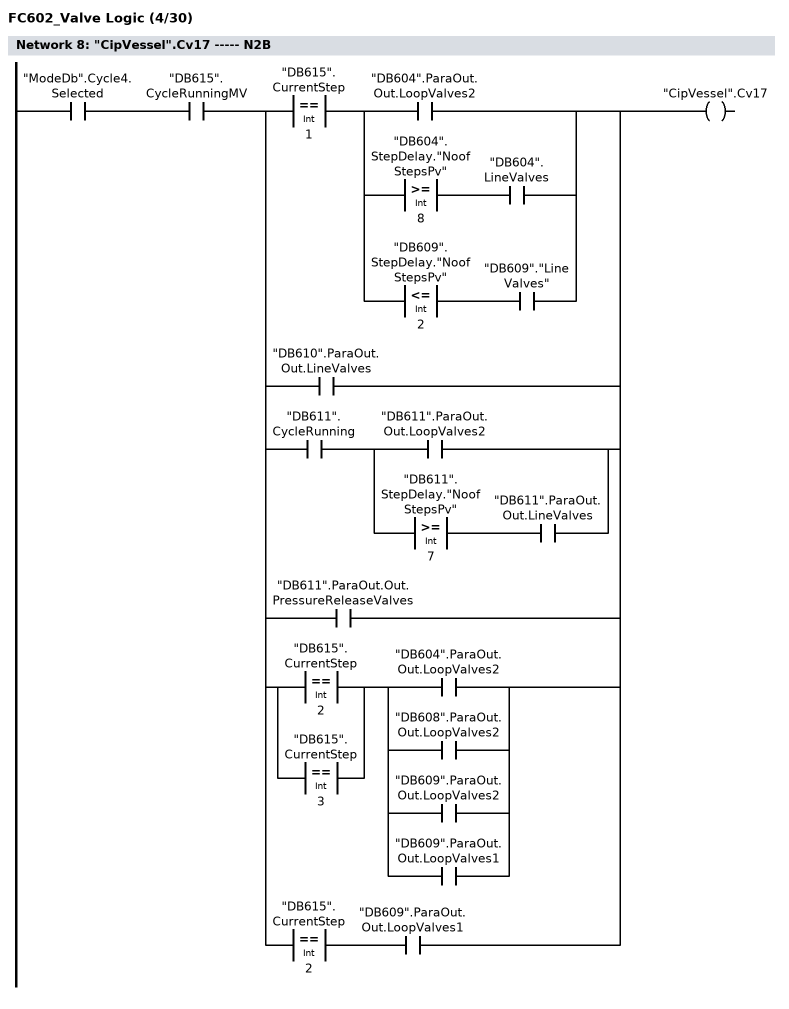
   RUNG wire#powerrail
      Contact( "ModeDb".Cycle4.Selected )
      Contact( "DB615".CycleRunningMV )
      wire#w1
      { S7_Templates := "SrcType := Int" } EQ_Contact(in1 := "DB615".CurrentStep, in2 := 1)
      wire#w2
      Contact( "DB604".ParaOut.Out.LoopValves2 )
      wire#w3
      Coil( "CipVessel".Cv17 )
   END_RUNG
   RUNG wire#w2
      { S7_Templates := "SrcType := Int" } GE_Contact(in1 := "DB604".StepDelay."Noof StepsPv", in2 := 8)
      Contact( "DB604".LineValves )
   END_RUNG wire#w3
   RUNG wire#w2
      { S7_Templates := "SrcType := Int" } LE_Contact(in1 := "DB609".StepDelay."Noof StepsPv", in2 := 2)
      Contact( "DB609"."Line Valves" )
   END_RUNG wire#w3
   RUNG wire#w1
      Contact( "DB610".ParaOut.Out.LineValves )
   END_RUNG wire#w3
   RUNG wire#w1
      Contact( "DB611".CycleRunning )
      wire#w4
      Contact( "DB611".ParaOut.Out.LoopValves2 )
   END_RUNG wire#w3
   RUNG wire#w4
      { S7_Templates := "SrcType := Int" } GE_Contact(in1 := "DB611".StepDelay."Noof StepsPv", in2 := 7)
      Contact( "DB611".ParaOut.Out.LineValves )
   END_RUNG wire#w3
   RUNG wire#w1
      Contact( "DB611".ParaOut.Out.PressureReleaseValves )
   END_RUNG wire#w3
   RUNG wire#w1
      { S7_Templates := "SrcType := Int" } EQ_Contact(in1 := "DB615".CurrentStep, in2 := 2)
      wire#w5
      Contact( "DB604".ParaOut.Out.LoopValves2 )
   END_RUNG wire#w3
   RUNG wire#w1
      { S7_Templates := "SrcType := Int" } EQ_Contact(in1 := "DB615".CurrentStep, in2 := 3)
   END_RUNG wire#w5
   RUNG wire#w5
      Contact( "DB608".ParaOut.Out.LoopValves2 )
   END_RUNG wire#w3
   RUNG wire#w5
      Contact( "DB609".ParaOut.Out.LoopValves2 )
   END_RUNG wire#w3
   RUNG wire#w5
      Contact( "DB609".ParaOut.Out.LoopValves1 )
   END_RUNG wire#w3
   RUNG wire#w1
      { S7_Templates := "SrcType := Int" } EQ_Contact(in1 := "DB615".CurrentStep, in2 := 2)
      Contact( "DB609".ParaOut.Out.LoopValves1 )
   END_RUNG wire#w3
   // the same network as SCL:
   "CipVessel".Cv17 := "ModeDb".Cycle4.Selected AND "DB615".CycleRunningMV AND ((("DB615".CurrentStep = 1) AND ("DB604".ParaOut.Out.LoopValves2 OR (("DB604".StepDelay."Noof StepsPv" >= 8) AND "DB604".LineValves) OR (("DB609".StepDelay."Noof StepsPv" <= 2) AND "DB609"."Line Valves"))) OR "DB610".ParaOut.Out.LineValves OR ("DB611".CycleRunning AND ("DB611".ParaOut.Out.LoopValves2 OR (("DB611".StepDelay."Noof StepsPv" >= 7) AND "DB611".ParaOut.Out.LineValves))) OR "DB611".ParaOut.Out.PressureReleaseValves OR ((("DB615".CurrentStep = 2) OR ("DB615".CurrentStep = 3)) AND ("DB604".ParaOut.Out.LoopValves2 OR "DB608".ParaOut.Out.LoopValves2 OR "DB609".ParaOut.Out.LoopValves2 OR "DB609".ParaOut.Out.LoopValves1)) OR (("DB615".CurrentStep = 2) AND "DB609".ParaOut.Out.LoopValves1));
END_REGION

REGION Network 9: "CipVessel".Cv16 ----- N2B
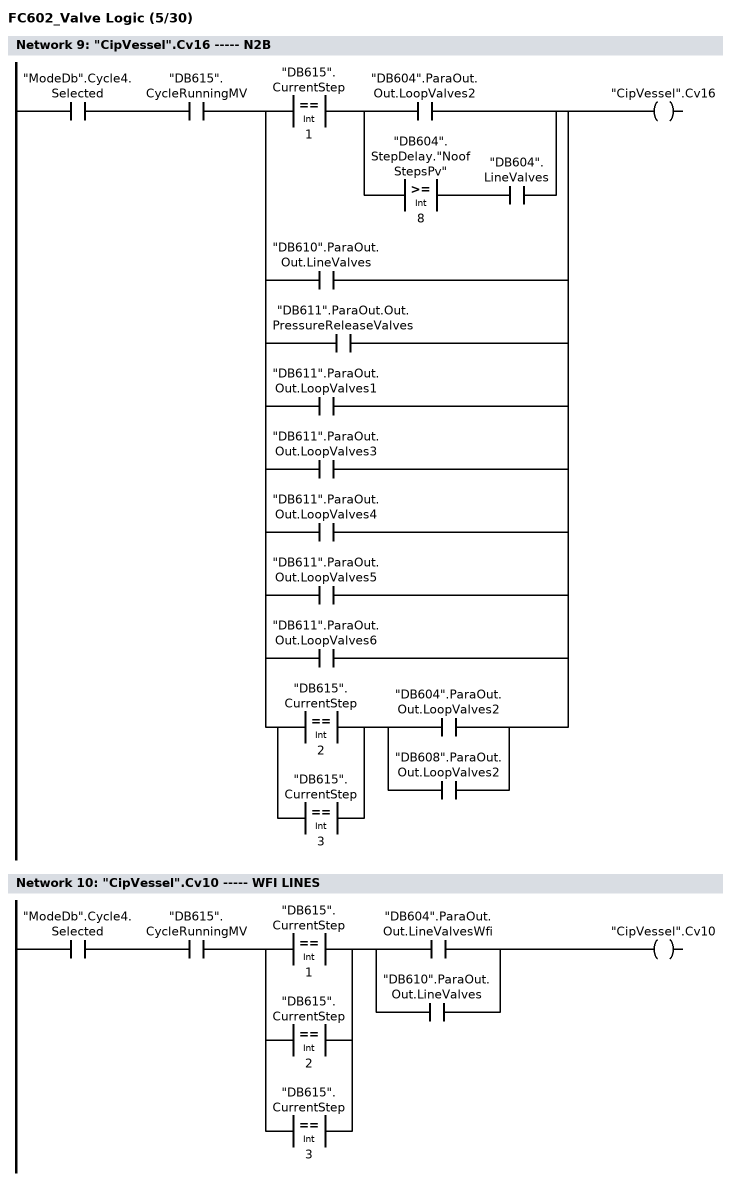
   RUNG wire#powerrail
      Contact( "ModeDb".Cycle4.Selected )
      Contact( "DB615".CycleRunningMV )
      wire#w1
      { S7_Templates := "SrcType := Int" } EQ_Contact(in1 := "DB615".CurrentStep, in2 := 1)
      wire#w2
      Contact( "DB604".ParaOut.Out.LoopValves2 )
      wire#w3
      Coil( "CipVessel".Cv16 )
   END_RUNG
   RUNG wire#w2
      { S7_Templates := "SrcType := Int" } GE_Contact(in1 := "DB604".StepDelay."Noof StepsPv", in2 := 8)
      Contact( "DB604".LineValves )
   END_RUNG wire#w3
   RUNG wire#w1
      Contact( "DB610".ParaOut.Out.LineValves )
   END_RUNG wire#w3
   RUNG wire#w1
      Contact( "DB611".ParaOut.Out.PressureReleaseValves )
   END_RUNG wire#w3
   RUNG wire#w1
      Contact( "DB611".ParaOut.Out.LoopValves1 )
   END_RUNG wire#w3
   RUNG wire#w1
      Contact( "DB611".ParaOut.Out.LoopValves3 )
   END_RUNG wire#w3
   RUNG wire#w1
      Contact( "DB611".ParaOut.Out.LoopValves4 )
   END_RUNG wire#w3
   RUNG wire#w1
      Contact( "DB611".ParaOut.Out.LoopValves5 )
   END_RUNG wire#w3
   RUNG wire#w1
      Contact( "DB611".ParaOut.Out.LoopValves6 )
   END_RUNG wire#w3
   RUNG wire#w1
      { S7_Templates := "SrcType := Int" } EQ_Contact(in1 := "DB615".CurrentStep, in2 := 2)
      wire#w4
      Contact( "DB604".ParaOut.Out.LoopValves2 )
   END_RUNG wire#w3
   RUNG wire#w1
      { S7_Templates := "SrcType := Int" } EQ_Contact(in1 := "DB615".CurrentStep, in2 := 3)
   END_RUNG wire#w4
   RUNG wire#w4
      Contact( "DB608".ParaOut.Out.LoopValves2 )
   END_RUNG wire#w3
   // the same network as SCL:
   "CipVessel".Cv16 := "ModeDb".Cycle4.Selected AND "DB615".CycleRunningMV AND ((("DB615".CurrentStep = 1) AND ("DB604".ParaOut.Out.LoopValves2 OR (("DB604".StepDelay."Noof StepsPv" >= 8) AND "DB604".LineValves))) OR "DB610".ParaOut.Out.LineValves OR "DB611".ParaOut.Out.PressureReleaseValves OR "DB611".ParaOut.Out.LoopValves1 OR "DB611".ParaOut.Out.LoopValves3 OR "DB611".ParaOut.Out.LoopValves4 OR "DB611".ParaOut.Out.LoopValves5 OR "DB611".ParaOut.Out.LoopValves6 OR ((("DB615".CurrentStep = 2) OR ("DB615".CurrentStep = 3)) AND ("DB604".ParaOut.Out.LoopValves2 OR "DB608".ParaOut.Out.LoopValves2)));
END_REGION

REGION Network 10: "CipVessel".Cv10 ----- WFI LINES
   RUNG wire#powerrail
      Contact( "ModeDb".Cycle4.Selected )
      Contact( "DB615".CycleRunningMV )
      wire#w1
      { S7_Templates := "SrcType := Int" } EQ_Contact(in1 := "DB615".CurrentStep, in2 := 1)
      wire#w2
      Contact( "DB604".ParaOut.Out.LineValvesWfi )
      wire#w3
      Coil( "CipVessel".Cv10 )
   END_RUNG
   RUNG wire#w1
      { S7_Templates := "SrcType := Int" } EQ_Contact(in1 := "DB615".CurrentStep, in2 := 2)
   END_RUNG wire#w2
   RUNG wire#w1
      { S7_Templates := "SrcType := Int" } EQ_Contact(in1 := "DB615".CurrentStep, in2 := 3)
   END_RUNG wire#w2
   RUNG wire#w2
      Contact( "DB610".ParaOut.Out.LineValves )
   END_RUNG wire#w3
   // the same network as SCL:
   "CipVessel".Cv10 := "ModeDb".Cycle4.Selected AND "DB615".CycleRunningMV AND (("DB615".CurrentStep = 1) OR ("DB615".CurrentStep = 2) OR ("DB615".CurrentStep = 3)) AND ("DB604".ParaOut.Out.LineValvesWfi OR "DB610".ParaOut.Out.LineValves);
END_REGION

REGION Network 11: "CipVessel".Cv15 ----- WFI LINES
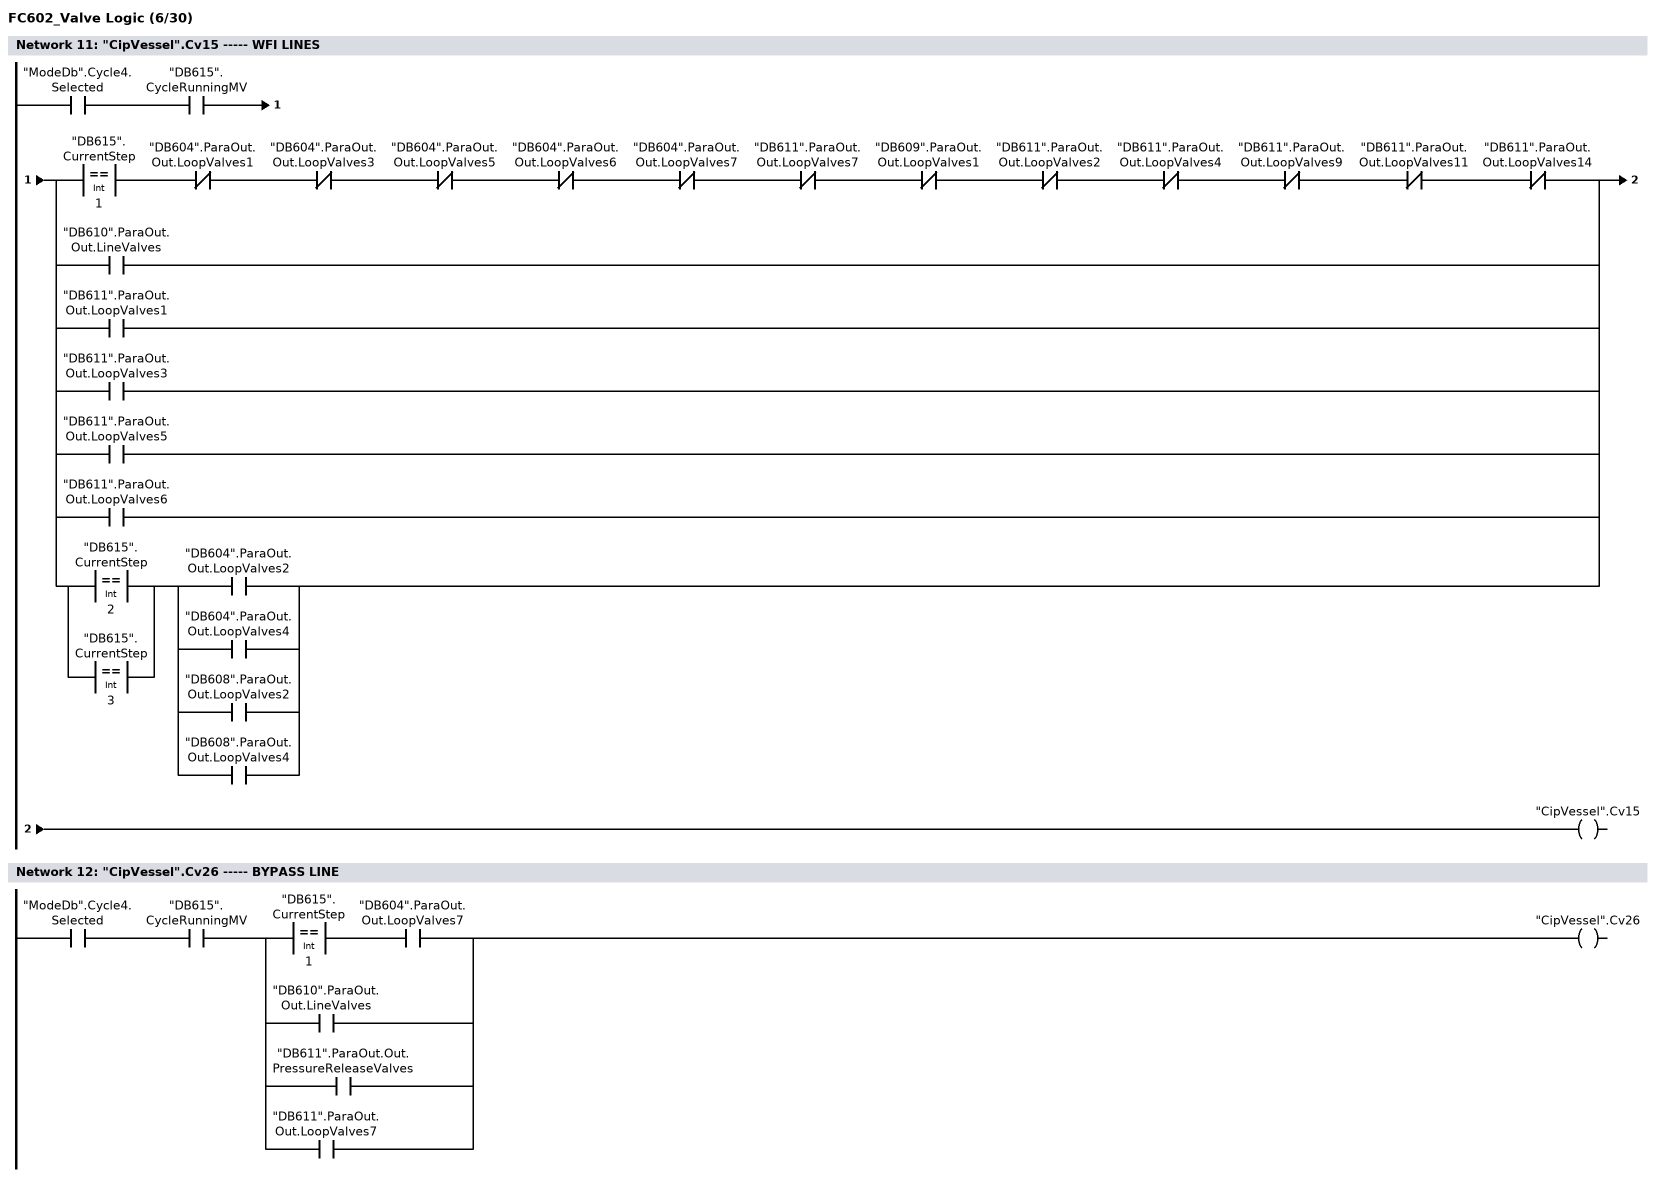
   RUNG wire#powerrail
      Contact( "ModeDb".Cycle4.Selected )
      Contact( "DB615".CycleRunningMV )
      wire#w1
      { S7_Templates := "SrcType := Int" } EQ_Contact(in1 := "DB615".CurrentStep, in2 := 1)
      I_Contact( "DB604".ParaOut.Out.LoopValves1 )
      I_Contact( "DB604".ParaOut.Out.LoopValves3 )
      I_Contact( "DB604".ParaOut.Out.LoopValves5 )
      I_Contact( "DB604".ParaOut.Out.LoopValves6 )
      I_Contact( "DB604".ParaOut.Out.LoopValves7 )
      I_Contact( "DB611".ParaOut.Out.LoopValves7 )
      I_Contact( "DB609".ParaOut.Out.LoopValves1 )
      I_Contact( "DB611".ParaOut.Out.LoopValves2 )
      I_Contact( "DB611".ParaOut.Out.LoopValves4 )
      I_Contact( "DB611".ParaOut.Out.LoopValves9 )
      I_Contact( "DB611".ParaOut.Out.LoopValves11 )
      I_Contact( "DB611".ParaOut.Out.LoopValves14 )
      wire#w2
      Coil( "CipVessel".Cv15 )
   END_RUNG
   RUNG wire#w1
      Contact( "DB610".ParaOut.Out.LineValves )
   END_RUNG wire#w2
   RUNG wire#w1
      Contact( "DB611".ParaOut.Out.LoopValves1 )
   END_RUNG wire#w2
   RUNG wire#w1
      Contact( "DB611".ParaOut.Out.LoopValves3 )
   END_RUNG wire#w2
   RUNG wire#w1
      Contact( "DB611".ParaOut.Out.LoopValves5 )
   END_RUNG wire#w2
   RUNG wire#w1
      Contact( "DB611".ParaOut.Out.LoopValves6 )
   END_RUNG wire#w2
   RUNG wire#w1
      { S7_Templates := "SrcType := Int" } EQ_Contact(in1 := "DB615".CurrentStep, in2 := 2)
      wire#w3
      Contact( "DB604".ParaOut.Out.LoopValves2 )
   END_RUNG wire#w2
   RUNG wire#w1
      { S7_Templates := "SrcType := Int" } EQ_Contact(in1 := "DB615".CurrentStep, in2 := 3)
   END_RUNG wire#w3
   RUNG wire#w3
      Contact( "DB604".ParaOut.Out.LoopValves4 )
   END_RUNG wire#w2
   RUNG wire#w3
      Contact( "DB608".ParaOut.Out.LoopValves2 )
   END_RUNG wire#w2
   RUNG wire#w3
      Contact( "DB608".ParaOut.Out.LoopValves4 )
   END_RUNG wire#w2
   // the same network as SCL:
   "CipVessel".Cv15 := "ModeDb".Cycle4.Selected AND "DB615".CycleRunningMV AND ((("DB615".CurrentStep = 1) AND NOT "DB604".ParaOut.Out.LoopValves1 AND NOT "DB604".ParaOut.Out.LoopValves3 AND NOT "DB604".ParaOut.Out.LoopValves5 AND NOT "DB604".ParaOut.Out.LoopValves6 AND NOT "DB604".ParaOut.Out.LoopValves7 AND NOT "DB611".ParaOut.Out.LoopValves7 AND NOT "DB609".ParaOut.Out.LoopValves1 AND NOT "DB611".ParaOut.Out.LoopValves2 AND NOT "DB611".ParaOut.Out.LoopValves4 AND NOT "DB611".ParaOut.Out.LoopValves9 AND NOT "DB611".ParaOut.Out.LoopValves11 AND NOT "DB611".ParaOut.Out.LoopValves14) OR "DB610".ParaOut.Out.LineValves OR "DB611".ParaOut.Out.LoopValves1 OR "DB611".ParaOut.Out.LoopValves3 OR "DB611".ParaOut.Out.LoopValves5 OR "DB611".ParaOut.Out.LoopValves6 OR ((("DB615".CurrentStep = 2) OR ("DB615".CurrentStep = 3)) AND ("DB604".ParaOut.Out.LoopValves2 OR "DB604".ParaOut.Out.LoopValves4 OR "DB608".ParaOut.Out.LoopValves2 OR "DB608".ParaOut.Out.LoopValves4)));
END_REGION

REGION Network 12: "CipVessel".Cv26 ----- BYPASS LINE
   RUNG wire#powerrail
      Contact( "ModeDb".Cycle4.Selected )
      Contact( "DB615".CycleRunningMV )
      wire#w1
      { S7_Templates := "SrcType := Int" } EQ_Contact(in1 := "DB615".CurrentStep, in2 := 1)
      Contact( "DB604".ParaOut.Out.LoopValves7 )
      wire#w2
      Coil( "CipVessel".Cv26 )
   END_RUNG
   RUNG wire#w1
      Contact( "DB610".ParaOut.Out.LineValves )
   END_RUNG wire#w2
   RUNG wire#w1
      Contact( "DB611".ParaOut.Out.PressureReleaseValves )
   END_RUNG wire#w2
   RUNG wire#w1
      Contact( "DB611".ParaOut.Out.LoopValves7 )
   END_RUNG wire#w2
   // the same network as SCL:
   "CipVessel".Cv26 := "ModeDb".Cycle4.Selected AND "DB615".CycleRunningMV AND ((("DB615".CurrentStep = 1) AND "DB604".ParaOut.Out.LoopValves7) OR "DB610".ParaOut.Out.LineValves OR "DB611".ParaOut.Out.PressureReleaseValves OR "DB611".ParaOut.Out.LoopValves7);
END_REGION

REGION Network 13: ------------- SAMPLING LINE ------------
END_REGION

REGION Network 14: "CipVessel".Cv12 - Sampling line
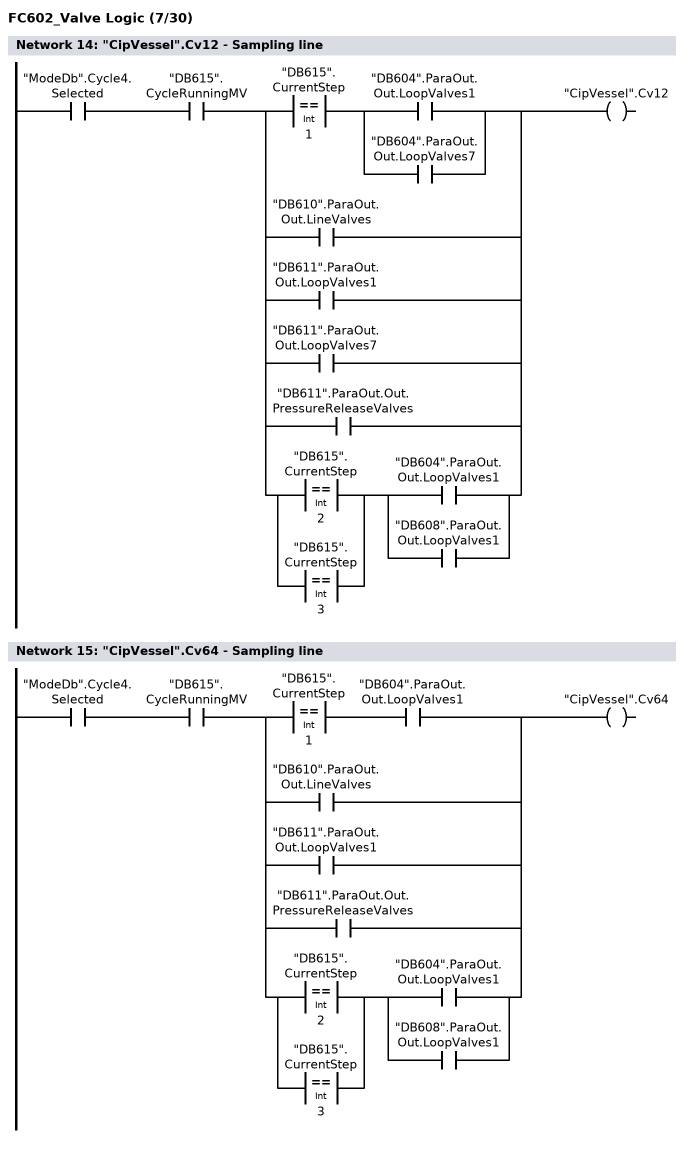
   RUNG wire#powerrail
      Contact( "ModeDb".Cycle4.Selected )
      Contact( "DB615".CycleRunningMV )
      wire#w1
      { S7_Templates := "SrcType := Int" } EQ_Contact(in1 := "DB615".CurrentStep, in2 := 1)
      wire#w2
      Contact( "DB604".ParaOut.Out.LoopValves1 )
      wire#w3
      Coil( "CipVessel".Cv12 )
   END_RUNG
   RUNG wire#w2
      Contact( "DB604".ParaOut.Out.LoopValves7 )
   END_RUNG wire#w3
   RUNG wire#w1
      Contact( "DB610".ParaOut.Out.LineValves )
   END_RUNG wire#w3
   RUNG wire#w1
      Contact( "DB611".ParaOut.Out.LoopValves1 )
   END_RUNG wire#w3
   RUNG wire#w1
      Contact( "DB611".ParaOut.Out.LoopValves7 )
   END_RUNG wire#w3
   RUNG wire#w1
      Contact( "DB611".ParaOut.Out.PressureReleaseValves )
   END_RUNG wire#w3
   RUNG wire#w1
      { S7_Templates := "SrcType := Int" } EQ_Contact(in1 := "DB615".CurrentStep, in2 := 2)
      wire#w4
      Contact( "DB604".ParaOut.Out.LoopValves1 )
   END_RUNG wire#w3
   RUNG wire#w1
      { S7_Templates := "SrcType := Int" } EQ_Contact(in1 := "DB615".CurrentStep, in2 := 3)
   END_RUNG wire#w4
   RUNG wire#w4
      Contact( "DB608".ParaOut.Out.LoopValves1 )
   END_RUNG wire#w3
   // the same network as SCL:
   "CipVessel".Cv12 := "ModeDb".Cycle4.Selected AND "DB615".CycleRunningMV AND ((("DB615".CurrentStep = 1) AND ("DB604".ParaOut.Out.LoopValves1 OR "DB604".ParaOut.Out.LoopValves7)) OR "DB610".ParaOut.Out.LineValves OR "DB611".ParaOut.Out.LoopValves1 OR "DB611".ParaOut.Out.LoopValves7 OR "DB611".ParaOut.Out.PressureReleaseValves OR ((("DB615".CurrentStep = 2) OR ("DB615".CurrentStep = 3)) AND ("DB604".ParaOut.Out.LoopValves1 OR "DB608".ParaOut.Out.LoopValves1)));
END_REGION

REGION Network 15: "CipVessel".Cv64 - Sampling line
   RUNG wire#powerrail
      Contact( "ModeDb".Cycle4.Selected )
      Contact( "DB615".CycleRunningMV )
      wire#w1
      { S7_Templates := "SrcType := Int" } EQ_Contact(in1 := "DB615".CurrentStep, in2 := 1)
      Contact( "DB604".ParaOut.Out.LoopValves1 )
      wire#w2
      Coil( "CipVessel".Cv64 )
   END_RUNG
   RUNG wire#w1
      Contact( "DB610".ParaOut.Out.LineValves )
   END_RUNG wire#w2
   RUNG wire#w1
      Contact( "DB611".ParaOut.Out.LoopValves1 )
   END_RUNG wire#w2
   RUNG wire#w1
      Contact( "DB611".ParaOut.Out.PressureReleaseValves )
   END_RUNG wire#w2
   RUNG wire#w1
      { S7_Templates := "SrcType := Int" } EQ_Contact(in1 := "DB615".CurrentStep, in2 := 2)
      wire#w3
      Contact( "DB604".ParaOut.Out.LoopValves1 )
   END_RUNG wire#w2
   RUNG wire#w1
      { S7_Templates := "SrcType := Int" } EQ_Contact(in1 := "DB615".CurrentStep, in2 := 3)
   END_RUNG wire#w3
   RUNG wire#w3
      Contact( "DB608".ParaOut.Out.LoopValves1 )
   END_RUNG wire#w2
   // the same network as SCL:
   "CipVessel".Cv64 := "ModeDb".Cycle4.Selected AND "DB615".CycleRunningMV AND ((("DB615".CurrentStep = 1) AND "DB604".ParaOut.Out.LoopValves1) OR "DB610".ParaOut.Out.LineValves OR "DB611".ParaOut.Out.LoopValves1 OR "DB611".ParaOut.Out.PressureReleaseValves OR ((("DB615".CurrentStep = 2) OR ("DB615".CurrentStep = 3)) AND ("DB604".ParaOut.Out.LoopValves1 OR "DB608".ParaOut.Out.LoopValves1)));
END_REGION

REGION Network 16: "CipVessel".Cv27 - Sampling line
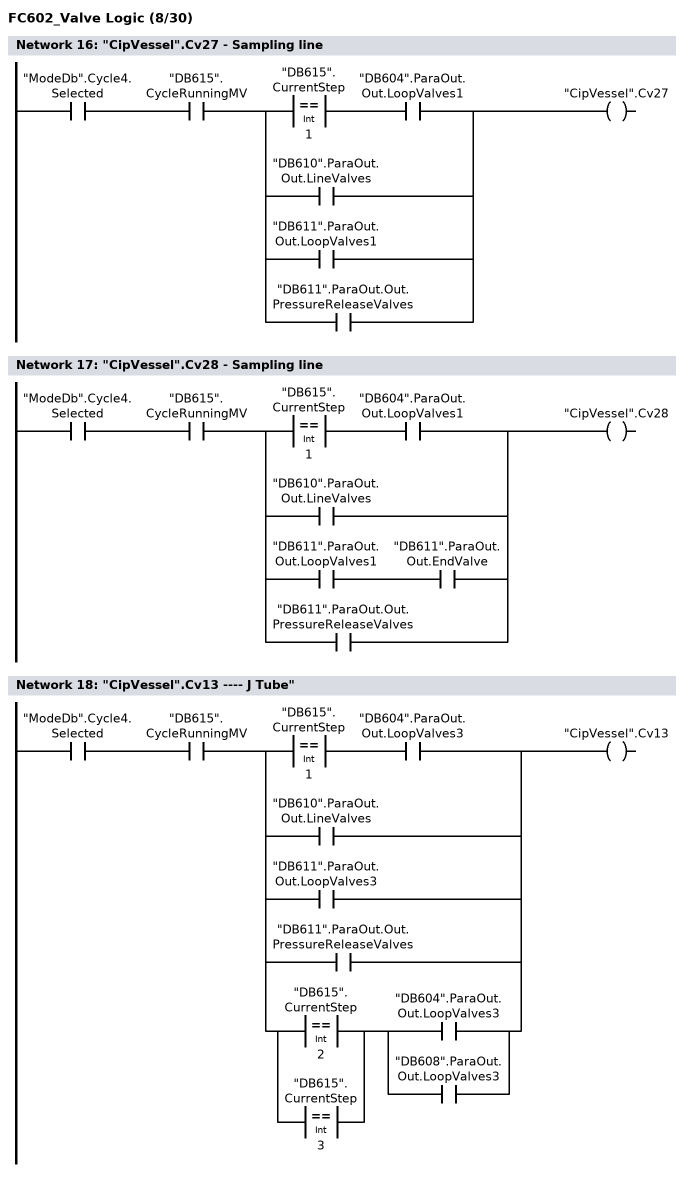
   RUNG wire#powerrail
      Contact( "ModeDb".Cycle4.Selected )
      Contact( "DB615".CycleRunningMV )
      wire#w1
      { S7_Templates := "SrcType := Int" } EQ_Contact(in1 := "DB615".CurrentStep, in2 := 1)
      Contact( "DB604".ParaOut.Out.LoopValves1 )
      wire#w2
      Coil( "CipVessel".Cv27 )
   END_RUNG
   RUNG wire#w1
      Contact( "DB610".ParaOut.Out.LineValves )
   END_RUNG wire#w2
   RUNG wire#w1
      Contact( "DB611".ParaOut.Out.LoopValves1 )
   END_RUNG wire#w2
   RUNG wire#w1
      Contact( "DB611".ParaOut.Out.PressureReleaseValves )
   END_RUNG wire#w2
   // the same network as SCL:
   "CipVessel".Cv27 := "ModeDb".Cycle4.Selected AND "DB615".CycleRunningMV AND ((("DB615".CurrentStep = 1) AND "DB604".ParaOut.Out.LoopValves1) OR "DB610".ParaOut.Out.LineValves OR "DB611".ParaOut.Out.LoopValves1 OR "DB611".ParaOut.Out.PressureReleaseValves);
END_REGION

REGION Network 17: "CipVessel".Cv28 - Sampling line
   RUNG wire#powerrail
      Contact( "ModeDb".Cycle4.Selected )
      Contact( "DB615".CycleRunningMV )
      wire#w1
      { S7_Templates := "SrcType := Int" } EQ_Contact(in1 := "DB615".CurrentStep, in2 := 1)
      Contact( "DB604".ParaOut.Out.LoopValves1 )
      wire#w2
      Coil( "CipVessel".Cv28 )
   END_RUNG
   RUNG wire#w1
      Contact( "DB610".ParaOut.Out.LineValves )
   END_RUNG wire#w2
   RUNG wire#w1
      Contact( "DB611".ParaOut.Out.LoopValves1 )
      Contact( "DB611".ParaOut.Out.EndValve )
   END_RUNG wire#w2
   RUNG wire#w1
      Contact( "DB611".ParaOut.Out.PressureReleaseValves )
   END_RUNG wire#w2
   // the same network as SCL:
   "CipVessel".Cv28 := "ModeDb".Cycle4.Selected AND "DB615".CycleRunningMV AND ((("DB615".CurrentStep = 1) AND "DB604".ParaOut.Out.LoopValves1) OR "DB610".ParaOut.Out.LineValves OR ("DB611".ParaOut.Out.LoopValves1 AND "DB611".ParaOut.Out.EndValve) OR "DB611".ParaOut.Out.PressureReleaseValves);
END_REGION

REGION Network 18: "CipVessel".Cv13 ---- J Tube"
   RUNG wire#powerrail
      Contact( "ModeDb".Cycle4.Selected )
      Contact( "DB615".CycleRunningMV )
      wire#w1
      { S7_Templates := "SrcType := Int" } EQ_Contact(in1 := "DB615".CurrentStep, in2 := 1)
      Contact( "DB604".ParaOut.Out.LoopValves3 )
      wire#w2
      Coil( "CipVessel".Cv13 )
   END_RUNG
   RUNG wire#w1
      Contact( "DB610".ParaOut.Out.LineValves )
   END_RUNG wire#w2
   RUNG wire#w1
      Contact( "DB611".ParaOut.Out.LoopValves3 )
   END_RUNG wire#w2
   RUNG wire#w1
      Contact( "DB611".ParaOut.Out.PressureReleaseValves )
   END_RUNG wire#w2
   RUNG wire#w1
      { S7_Templates := "SrcType := Int" } EQ_Contact(in1 := "DB615".CurrentStep, in2 := 2)
      wire#w3
      Contact( "DB604".ParaOut.Out.LoopValves3 )
   END_RUNG wire#w2
   RUNG wire#w1
      { S7_Templates := "SrcType := Int" } EQ_Contact(in1 := "DB615".CurrentStep, in2 := 3)
   END_RUNG wire#w3
   RUNG wire#w3
      Contact( "DB608".ParaOut.Out.LoopValves3 )
   END_RUNG wire#w2
   // the same network as SCL:
   "CipVessel".Cv13 := "ModeDb".Cycle4.Selected AND "DB615".CycleRunningMV AND ((("DB615".CurrentStep = 1) AND "DB604".ParaOut.Out.LoopValves3) OR "DB610".ParaOut.Out.LineValves OR "DB611".ParaOut.Out.LoopValves3 OR "DB611".ParaOut.Out.PressureReleaseValves OR ((("DB615".CurrentStep = 2) OR ("DB615".CurrentStep = 3)) AND ("DB604".ParaOut.Out.LoopValves3 OR "DB608".ParaOut.Out.LoopValves3)));
END_REGION

REGION Network 19: "CipVessel".Cv63 ---- N2S
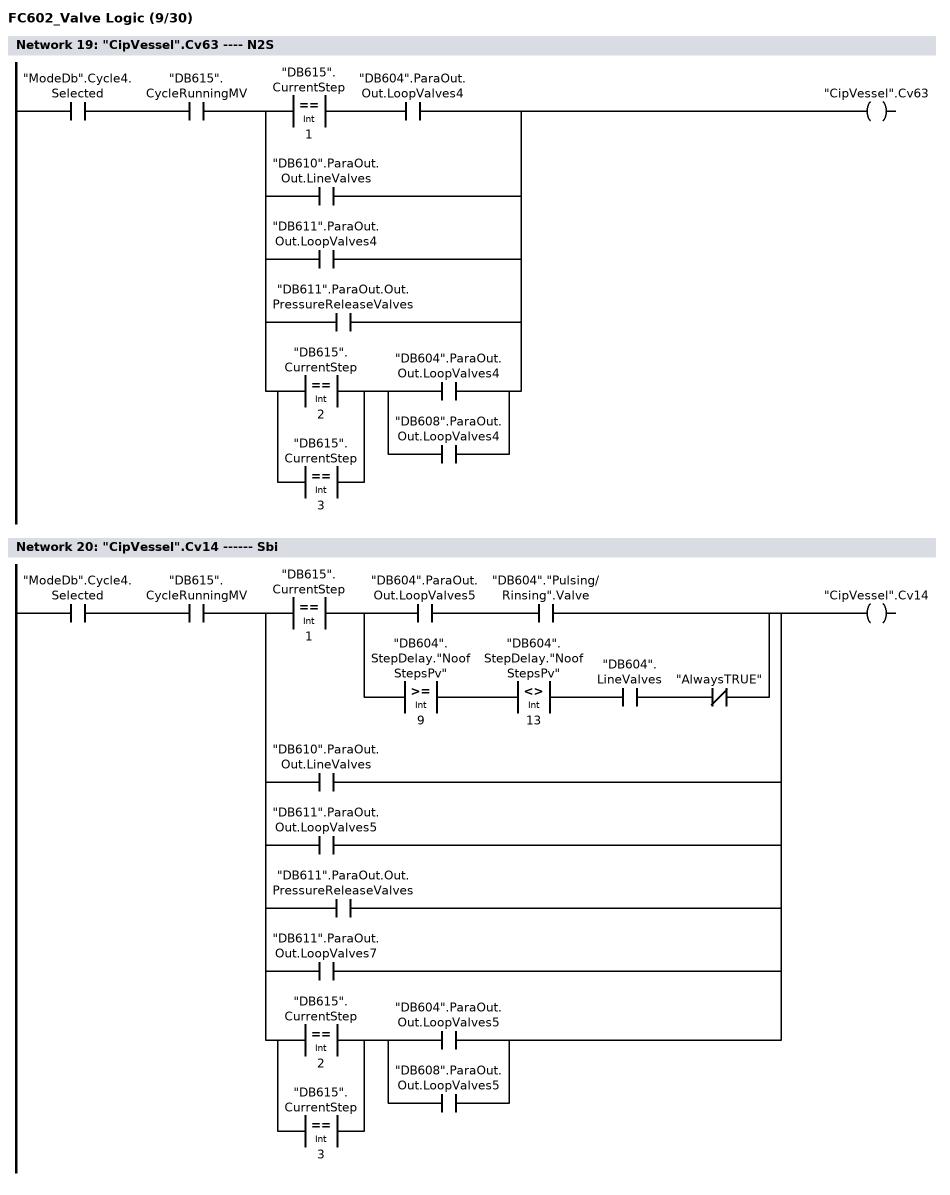
   RUNG wire#powerrail
      Contact( "ModeDb".Cycle4.Selected )
      Contact( "DB615".CycleRunningMV )
      wire#w1
      { S7_Templates := "SrcType := Int" } EQ_Contact(in1 := "DB615".CurrentStep, in2 := 1)
      Contact( "DB604".ParaOut.Out.LoopValves4 )
      wire#w2
      Coil( "CipVessel".Cv63 )
   END_RUNG
   RUNG wire#w1
      Contact( "DB610".ParaOut.Out.LineValves )
   END_RUNG wire#w2
   RUNG wire#w1
      Contact( "DB611".ParaOut.Out.LoopValves4 )
   END_RUNG wire#w2
   RUNG wire#w1
      Contact( "DB611".ParaOut.Out.PressureReleaseValves )
   END_RUNG wire#w2
   RUNG wire#w1
      { S7_Templates := "SrcType := Int" } EQ_Contact(in1 := "DB615".CurrentStep, in2 := 2)
      wire#w3
      Contact( "DB604".ParaOut.Out.LoopValves4 )
   END_RUNG wire#w2
   RUNG wire#w1
      { S7_Templates := "SrcType := Int" } EQ_Contact(in1 := "DB615".CurrentStep, in2 := 3)
   END_RUNG wire#w3
   RUNG wire#w3
      Contact( "DB608".ParaOut.Out.LoopValves4 )
   END_RUNG wire#w2
   // the same network as SCL:
   "CipVessel".Cv63 := "ModeDb".Cycle4.Selected AND "DB615".CycleRunningMV AND ((("DB615".CurrentStep = 1) AND "DB604".ParaOut.Out.LoopValves4) OR "DB610".ParaOut.Out.LineValves OR "DB611".ParaOut.Out.LoopValves4 OR "DB611".ParaOut.Out.PressureReleaseValves OR ((("DB615".CurrentStep = 2) OR ("DB615".CurrentStep = 3)) AND ("DB604".ParaOut.Out.LoopValves4 OR "DB608".ParaOut.Out.LoopValves4)));
END_REGION

REGION Network 20: "CipVessel".Cv14 ------ Sbi
   RUNG wire#powerrail
      Contact( "ModeDb".Cycle4.Selected )
      Contact( "DB615".CycleRunningMV )
      wire#w1
      { S7_Templates := "SrcType := Int" } EQ_Contact(in1 := "DB615".CurrentStep, in2 := 1)
      wire#w2
      Contact( "DB604".ParaOut.Out.LoopValves5 )
      Contact( "DB604"."Pulsing/Rinsing".Valve )
      wire#w3
      Coil( "CipVessel".Cv14 )
   END_RUNG
   RUNG wire#w2
      { S7_Templates := "SrcType := Int" } GE_Contact(in1 := "DB604".StepDelay."Noof StepsPv", in2 := 9)
      { S7_Templates := "SrcType := Int" } NE_Contact(in1 := "DB604".StepDelay."Noof StepsPv", in2 := 13)
      Contact( "DB604".LineValves )
      I_Contact( "AlwaysTRUE" )
   END_RUNG wire#w3
   RUNG wire#w1
      Contact( "DB610".ParaOut.Out.LineValves )
   END_RUNG wire#w3
   RUNG wire#w1
      Contact( "DB611".ParaOut.Out.LoopValves5 )
   END_RUNG wire#w3
   RUNG wire#w1
      Contact( "DB611".ParaOut.Out.PressureReleaseValves )
   END_RUNG wire#w3
   RUNG wire#w1
      Contact( "DB611".ParaOut.Out.LoopValves7 )
   END_RUNG wire#w3
   RUNG wire#w1
      { S7_Templates := "SrcType := Int" } EQ_Contact(in1 := "DB615".CurrentStep, in2 := 2)
      wire#w4
      Contact( "DB604".ParaOut.Out.LoopValves5 )
   END_RUNG wire#w3
   RUNG wire#w1
      { S7_Templates := "SrcType := Int" } EQ_Contact(in1 := "DB615".CurrentStep, in2 := 3)
   END_RUNG wire#w4
   RUNG wire#w4
      Contact( "DB608".ParaOut.Out.LoopValves5 )
   END_RUNG wire#w3
   // the same network as SCL:
   "CipVessel".Cv14 := "ModeDb".Cycle4.Selected AND "DB615".CycleRunningMV AND ((("DB615".CurrentStep = 1) AND (("DB604".ParaOut.Out.LoopValves5 AND "DB604"."Pulsing/Rinsing".Valve) OR (("DB604".StepDelay."Noof StepsPv" >= 9) AND ("DB604".StepDelay."Noof StepsPv" <> 13) AND "DB604".LineValves AND NOT "AlwaysTRUE"))) OR "DB610".ParaOut.Out.LineValves OR "DB611".ParaOut.Out.LoopValves5 OR "DB611".ParaOut.Out.PressureReleaseValves OR "DB611".ParaOut.Out.LoopValves7 OR ((("DB615".CurrentStep = 2) OR ("DB615".CurrentStep = 3)) AND ("DB604".ParaOut.Out.LoopValves5 OR "DB608".ParaOut.Out.LoopValves5)));
END_REGION

REGION Network 21: "CipVessel".Fbov01 ------ Fbov
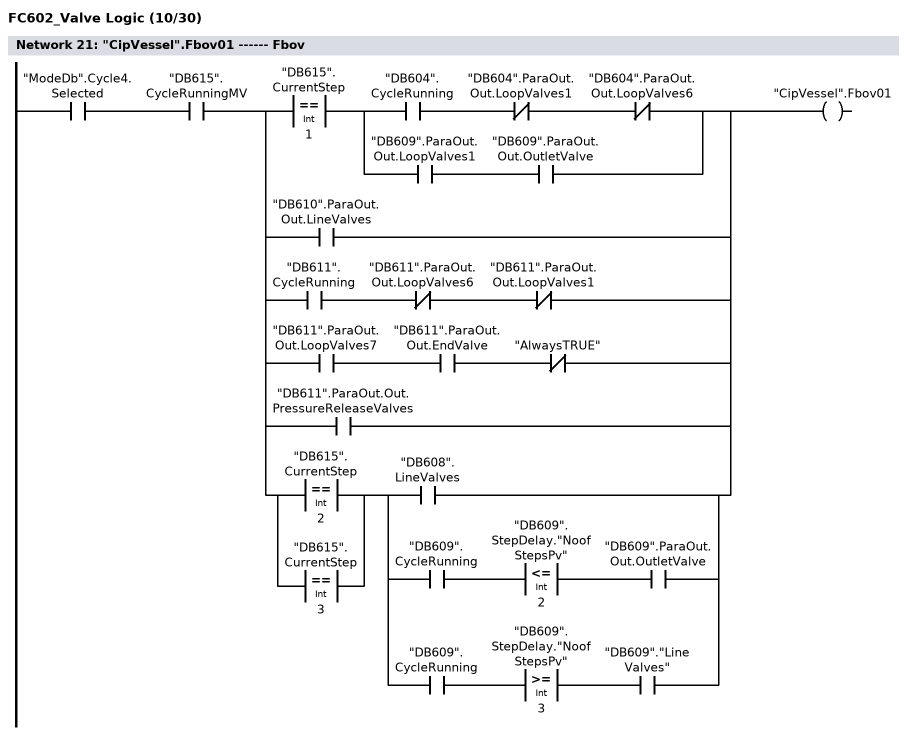
   RUNG wire#powerrail
      Contact( "ModeDb".Cycle4.Selected )
      Contact( "DB615".CycleRunningMV )
      wire#w1
      { S7_Templates := "SrcType := Int" } EQ_Contact(in1 := "DB615".CurrentStep, in2 := 1)
      wire#w2
      Contact( "DB604".CycleRunning )
      I_Contact( "DB604".ParaOut.Out.LoopValves1 )
      I_Contact( "DB604".ParaOut.Out.LoopValves6 )
      wire#w3
      Coil( "CipVessel".Fbov01 )
   END_RUNG
   RUNG wire#w2
      Contact( "DB609".ParaOut.Out.LoopValves1 )
      Contact( "DB609".ParaOut.Out.OutletValve )
   END_RUNG wire#w3
   RUNG wire#w1
      Contact( "DB610".ParaOut.Out.LineValves )
   END_RUNG wire#w3
   RUNG wire#w1
      Contact( "DB611".CycleRunning )
      I_Contact( "DB611".ParaOut.Out.LoopValves6 )
      I_Contact( "DB611".ParaOut.Out.LoopValves1 )
   END_RUNG wire#w3
   RUNG wire#w1
      Contact( "DB611".ParaOut.Out.LoopValves7 )
      Contact( "DB611".ParaOut.Out.EndValve )
      I_Contact( "AlwaysTRUE" )
   END_RUNG wire#w3
   RUNG wire#w1
      Contact( "DB611".ParaOut.Out.PressureReleaseValves )
   END_RUNG wire#w3
   RUNG wire#w1
      { S7_Templates := "SrcType := Int" } EQ_Contact(in1 := "DB615".CurrentStep, in2 := 2)
      wire#w4
      Contact( "DB608".LineValves )
   END_RUNG wire#w3
   RUNG wire#w1
      { S7_Templates := "SrcType := Int" } EQ_Contact(in1 := "DB615".CurrentStep, in2 := 3)
   END_RUNG wire#w4
   RUNG wire#w4
      Contact( "DB609".CycleRunning )
      { S7_Templates := "SrcType := Int" } LE_Contact(in1 := "DB609".StepDelay."Noof StepsPv", in2 := 2)
      Contact( "DB609".ParaOut.Out.OutletValve )
   END_RUNG wire#w3
   RUNG wire#w4
      Contact( "DB609".CycleRunning )
      { S7_Templates := "SrcType := Int" } GE_Contact(in1 := "DB609".StepDelay."Noof StepsPv", in2 := 3)
      Contact( "DB609"."Line Valves" )
   END_RUNG wire#w3
   // the same network as SCL:
   "CipVessel".Fbov01 := "ModeDb".Cycle4.Selected AND "DB615".CycleRunningMV AND ((("DB615".CurrentStep = 1) AND (("DB604".CycleRunning AND NOT "DB604".ParaOut.Out.LoopValves1 AND NOT "DB604".ParaOut.Out.LoopValves6) OR ("DB609".ParaOut.Out.LoopValves1 AND "DB609".ParaOut.Out.OutletValve))) OR "DB610".ParaOut.Out.LineValves OR ("DB611".CycleRunning AND NOT "DB611".ParaOut.Out.LoopValves6 AND NOT "DB611".ParaOut.Out.LoopValves1) OR ("DB611".ParaOut.Out.LoopValves7 AND "DB611".ParaOut.Out.EndValve AND NOT "AlwaysTRUE") OR "DB611".ParaOut.Out.PressureReleaseValves OR ((("DB615".CurrentStep = 2) OR ("DB615".CurrentStep = 3)) AND ("DB608".LineValves OR ("DB609".CycleRunning AND ("DB609".StepDelay."Noof StepsPv" <= 2) AND "DB609".ParaOut.Out.OutletValve) OR ("DB609".CycleRunning AND ("DB609".StepDelay."Noof StepsPv" >= 3) AND "DB609"."Line Valves"))));
END_REGION

REGION Network 22: ----------- VESSEL DRAIN LINE ------------
END_REGION

REGION Network 23: "CipVessel".Cv30
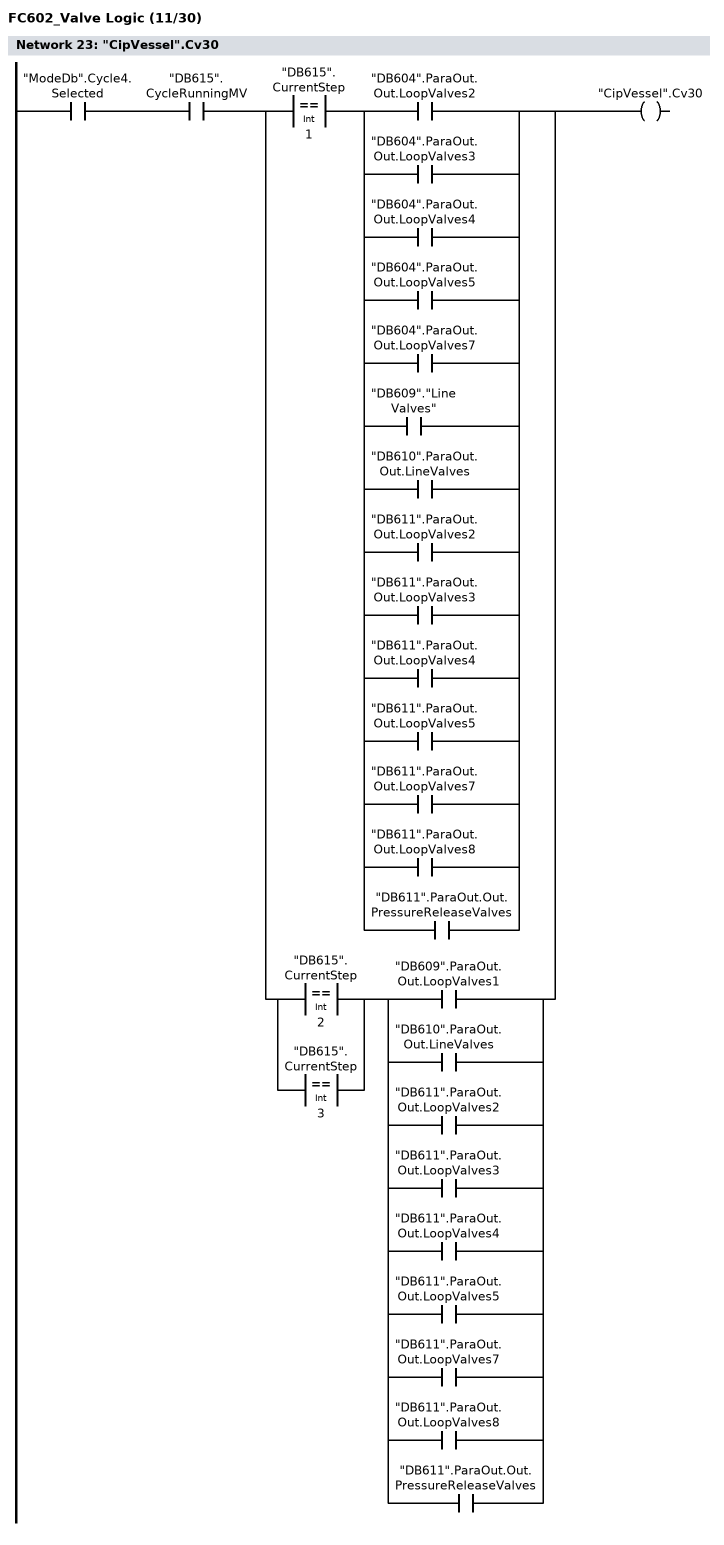
   RUNG wire#powerrail
      Contact( "ModeDb".Cycle4.Selected )
      Contact( "DB615".CycleRunningMV )
      wire#w1
      { S7_Templates := "SrcType := Int" } EQ_Contact(in1 := "DB615".CurrentStep, in2 := 1)
      wire#w2
      Contact( "DB604".ParaOut.Out.LoopValves2 )
      wire#w3
      Coil( "CipVessel".Cv30 )
   END_RUNG
   RUNG wire#w2
      Contact( "DB604".ParaOut.Out.LoopValves3 )
   END_RUNG wire#w3
   RUNG wire#w2
      Contact( "DB604".ParaOut.Out.LoopValves4 )
   END_RUNG wire#w3
   RUNG wire#w2
      Contact( "DB604".ParaOut.Out.LoopValves5 )
   END_RUNG wire#w3
   RUNG wire#w2
      Contact( "DB604".ParaOut.Out.LoopValves7 )
   END_RUNG wire#w3
   RUNG wire#w2
      Contact( "DB609"."Line Valves" )
   END_RUNG wire#w3
   RUNG wire#w2
      Contact( "DB610".ParaOut.Out.LineValves )
   END_RUNG wire#w3
   RUNG wire#w2
      Contact( "DB611".ParaOut.Out.LoopValves2 )
   END_RUNG wire#w3
   RUNG wire#w2
      Contact( "DB611".ParaOut.Out.LoopValves3 )
   END_RUNG wire#w3
   RUNG wire#w2
      Contact( "DB611".ParaOut.Out.LoopValves4 )
   END_RUNG wire#w3
   RUNG wire#w2
      Contact( "DB611".ParaOut.Out.LoopValves5 )
   END_RUNG wire#w3
   RUNG wire#w2
      Contact( "DB611".ParaOut.Out.LoopValves7 )
   END_RUNG wire#w3
   RUNG wire#w2
      Contact( "DB611".ParaOut.Out.LoopValves8 )
   END_RUNG wire#w3
   RUNG wire#w2
      Contact( "DB611".ParaOut.Out.PressureReleaseValves )
   END_RUNG wire#w3
   RUNG wire#w1
      { S7_Templates := "SrcType := Int" } EQ_Contact(in1 := "DB615".CurrentStep, in2 := 2)
      wire#w4
      Contact( "DB609".ParaOut.Out.LoopValves1 )
   END_RUNG wire#w3
   RUNG wire#w1
      { S7_Templates := "SrcType := Int" } EQ_Contact(in1 := "DB615".CurrentStep, in2 := 3)
   END_RUNG wire#w4
   RUNG wire#w4
      Contact( "DB610".ParaOut.Out.LineValves )
   END_RUNG wire#w3
   RUNG wire#w4
      Contact( "DB611".ParaOut.Out.LoopValves2 )
   END_RUNG wire#w3
   RUNG wire#w4
      Contact( "DB611".ParaOut.Out.LoopValves3 )
   END_RUNG wire#w3
   RUNG wire#w4
      Contact( "DB611".ParaOut.Out.LoopValves4 )
   END_RUNG wire#w3
   RUNG wire#w4
      Contact( "DB611".ParaOut.Out.LoopValves5 )
   END_RUNG wire#w3
   RUNG wire#w4
      Contact( "DB611".ParaOut.Out.LoopValves7 )
   END_RUNG wire#w3
   RUNG wire#w4
      Contact( "DB611".ParaOut.Out.LoopValves8 )
   END_RUNG wire#w3
   RUNG wire#w4
      Contact( "DB611".ParaOut.Out.PressureReleaseValves )
   END_RUNG wire#w3
   // the same network as SCL:
   "CipVessel".Cv30 := "ModeDb".Cycle4.Selected AND "DB615".CycleRunningMV AND ((("DB615".CurrentStep = 1) AND ("DB604".ParaOut.Out.LoopValves2 OR "DB604".ParaOut.Out.LoopValves3 OR "DB604".ParaOut.Out.LoopValves4 OR "DB604".ParaOut.Out.LoopValves5 OR "DB604".ParaOut.Out.LoopValves7 OR "DB609"."Line Valves" OR "DB610".ParaOut.Out.LineValves OR "DB611".ParaOut.Out.LoopValves2 OR "DB611".ParaOut.Out.LoopValves3 OR "DB611".ParaOut.Out.LoopValves4 OR "DB611".ParaOut.Out.LoopValves5 OR "DB611".ParaOut.Out.LoopValves7 OR "DB611".ParaOut.Out.LoopValves8 OR "DB611".ParaOut.Out.PressureReleaseValves)) OR ((("DB615".CurrentStep = 2) OR ("DB615".CurrentStep = 3)) AND ("DB609".ParaOut.Out.LoopValves1 OR "DB610".ParaOut.Out.LineValves OR "DB611".ParaOut.Out.LoopValves2 OR "DB611".ParaOut.Out.LoopValves3 OR "DB611".ParaOut.Out.LoopValves4 OR "DB611".ParaOut.Out.LoopValves5 OR "DB611".ParaOut.Out.LoopValves7 OR "DB611".ParaOut.Out.LoopValves8 OR "DB611".ParaOut.Out.PressureReleaseValves)));
END_REGION

REGION Network 24: "CipVessel".Cv33
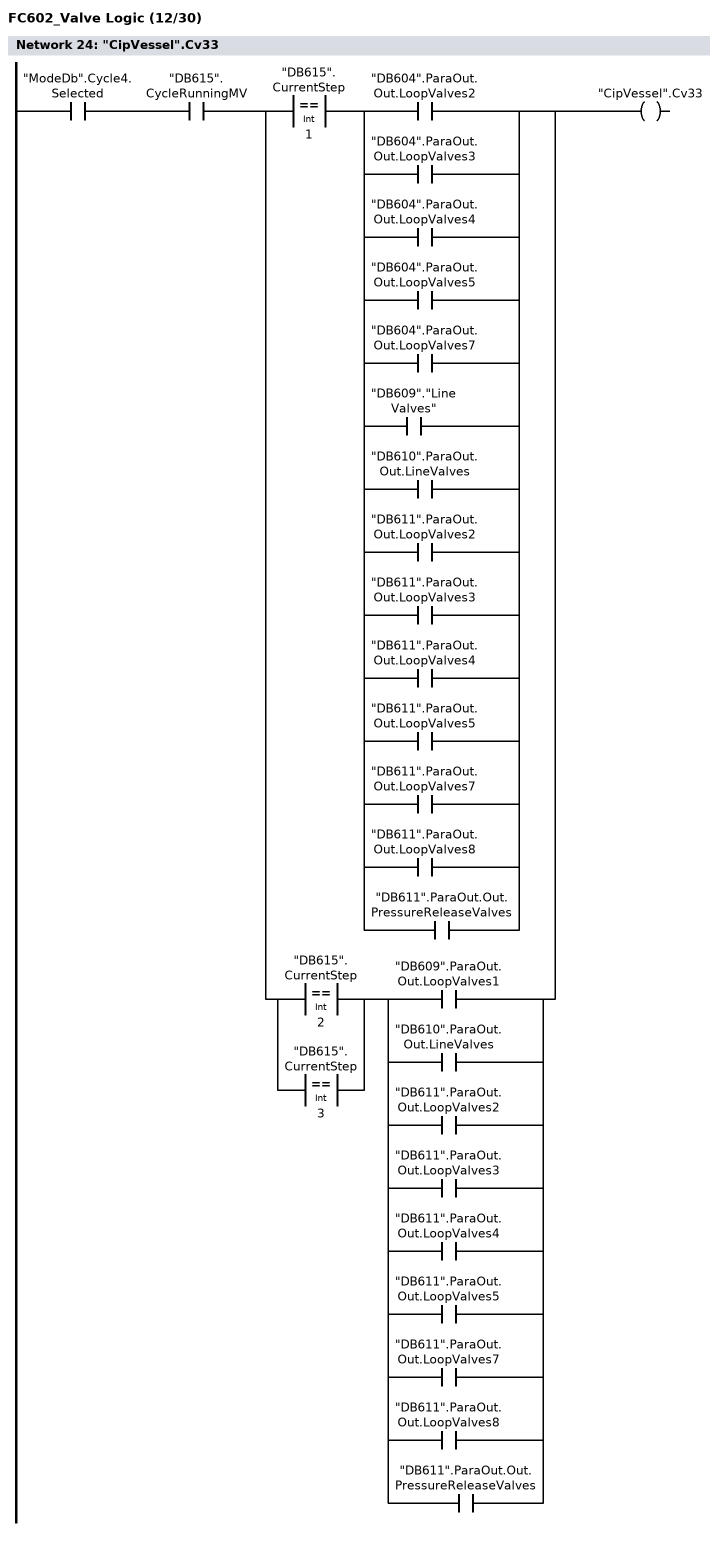
   RUNG wire#powerrail
      Contact( "ModeDb".Cycle4.Selected )
      Contact( "DB615".CycleRunningMV )
      wire#w1
      { S7_Templates := "SrcType := Int" } EQ_Contact(in1 := "DB615".CurrentStep, in2 := 1)
      wire#w2
      Contact( "DB604".ParaOut.Out.LoopValves2 )
      wire#w3
      Coil( "CipVessel".Cv33 )
   END_RUNG
   RUNG wire#w2
      Contact( "DB604".ParaOut.Out.LoopValves3 )
   END_RUNG wire#w3
   RUNG wire#w2
      Contact( "DB604".ParaOut.Out.LoopValves4 )
   END_RUNG wire#w3
   RUNG wire#w2
      Contact( "DB604".ParaOut.Out.LoopValves5 )
   END_RUNG wire#w3
   RUNG wire#w2
      Contact( "DB604".ParaOut.Out.LoopValves7 )
   END_RUNG wire#w3
   RUNG wire#w2
      Contact( "DB609"."Line Valves" )
   END_RUNG wire#w3
   RUNG wire#w2
      Contact( "DB610".ParaOut.Out.LineValves )
   END_RUNG wire#w3
   RUNG wire#w2
      Contact( "DB611".ParaOut.Out.LoopValves2 )
   END_RUNG wire#w3
   RUNG wire#w2
      Contact( "DB611".ParaOut.Out.LoopValves3 )
   END_RUNG wire#w3
   RUNG wire#w2
      Contact( "DB611".ParaOut.Out.LoopValves4 )
   END_RUNG wire#w3
   RUNG wire#w2
      Contact( "DB611".ParaOut.Out.LoopValves5 )
   END_RUNG wire#w3
   RUNG wire#w2
      Contact( "DB611".ParaOut.Out.LoopValves7 )
   END_RUNG wire#w3
   RUNG wire#w2
      Contact( "DB611".ParaOut.Out.LoopValves8 )
   END_RUNG wire#w3
   RUNG wire#w2
      Contact( "DB611".ParaOut.Out.PressureReleaseValves )
   END_RUNG wire#w3
   RUNG wire#w1
      { S7_Templates := "SrcType := Int" } EQ_Contact(in1 := "DB615".CurrentStep, in2 := 2)
      wire#w4
      Contact( "DB609".ParaOut.Out.LoopValves1 )
   END_RUNG wire#w3
   RUNG wire#w1
      { S7_Templates := "SrcType := Int" } EQ_Contact(in1 := "DB615".CurrentStep, in2 := 3)
   END_RUNG wire#w4
   RUNG wire#w4
      Contact( "DB610".ParaOut.Out.LineValves )
   END_RUNG wire#w3
   RUNG wire#w4
      Contact( "DB611".ParaOut.Out.LoopValves2 )
   END_RUNG wire#w3
   RUNG wire#w4
      Contact( "DB611".ParaOut.Out.LoopValves3 )
   END_RUNG wire#w3
   RUNG wire#w4
      Contact( "DB611".ParaOut.Out.LoopValves4 )
   END_RUNG wire#w3
   RUNG wire#w4
      Contact( "DB611".ParaOut.Out.LoopValves5 )
   END_RUNG wire#w3
   RUNG wire#w4
      Contact( "DB611".ParaOut.Out.LoopValves7 )
   END_RUNG wire#w3
   RUNG wire#w4
      Contact( "DB611".ParaOut.Out.LoopValves8 )
   END_RUNG wire#w3
   RUNG wire#w4
      Contact( "DB611".ParaOut.Out.PressureReleaseValves )
   END_RUNG wire#w3
   // the same network as SCL:
   "CipVessel".Cv33 := "ModeDb".Cycle4.Selected AND "DB615".CycleRunningMV AND ((("DB615".CurrentStep = 1) AND ("DB604".ParaOut.Out.LoopValves2 OR "DB604".ParaOut.Out.LoopValves3 OR "DB604".ParaOut.Out.LoopValves4 OR "DB604".ParaOut.Out.LoopValves5 OR "DB604".ParaOut.Out.LoopValves7 OR "DB609"."Line Valves" OR "DB610".ParaOut.Out.LineValves OR "DB611".ParaOut.Out.LoopValves2 OR "DB611".ParaOut.Out.LoopValves3 OR "DB611".ParaOut.Out.LoopValves4 OR "DB611".ParaOut.Out.LoopValves5 OR "DB611".ParaOut.Out.LoopValves7 OR "DB611".ParaOut.Out.LoopValves8 OR "DB611".ParaOut.Out.PressureReleaseValves)) OR ((("DB615".CurrentStep = 2) OR ("DB615".CurrentStep = 3)) AND ("DB609".ParaOut.Out.LoopValves1 OR "DB610".ParaOut.Out.LineValves OR "DB611".ParaOut.Out.LoopValves2 OR "DB611".ParaOut.Out.LoopValves3 OR "DB611".ParaOut.Out.LoopValves4 OR "DB611".ParaOut.Out.LoopValves5 OR "DB611".ParaOut.Out.LoopValves7 OR "DB611".ParaOut.Out.LoopValves8 OR "DB611".ParaOut.Out.PressureReleaseValves)));
END_REGION

REGION Network 25: "CipVessel".Cv34
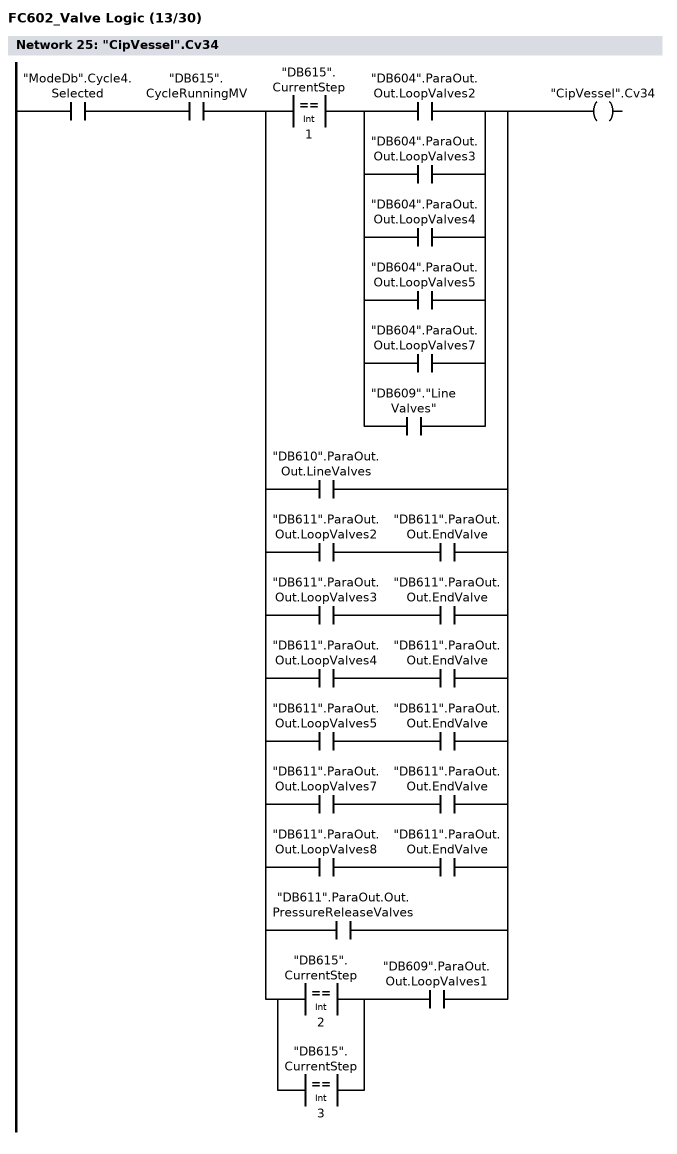
   RUNG wire#powerrail
      Contact( "ModeDb".Cycle4.Selected )
      Contact( "DB615".CycleRunningMV )
      wire#w1
      { S7_Templates := "SrcType := Int" } EQ_Contact(in1 := "DB615".CurrentStep, in2 := 1)
      wire#w2
      Contact( "DB604".ParaOut.Out.LoopValves2 )
      wire#w3
      Coil( "CipVessel".Cv34 )
   END_RUNG
   RUNG wire#w2
      Contact( "DB604".ParaOut.Out.LoopValves3 )
   END_RUNG wire#w3
   RUNG wire#w2
      Contact( "DB604".ParaOut.Out.LoopValves4 )
   END_RUNG wire#w3
   RUNG wire#w2
      Contact( "DB604".ParaOut.Out.LoopValves5 )
   END_RUNG wire#w3
   RUNG wire#w2
      Contact( "DB604".ParaOut.Out.LoopValves7 )
   END_RUNG wire#w3
   RUNG wire#w2
      Contact( "DB609"."Line Valves" )
   END_RUNG wire#w3
   RUNG wire#w1
      Contact( "DB610".ParaOut.Out.LineValves )
   END_RUNG wire#w3
   RUNG wire#w1
      Contact( "DB611".ParaOut.Out.LoopValves2 )
      Contact( "DB611".ParaOut.Out.EndValve )
   END_RUNG wire#w3
   RUNG wire#w1
      Contact( "DB611".ParaOut.Out.LoopValves3 )
      Contact( "DB611".ParaOut.Out.EndValve )
   END_RUNG wire#w3
   RUNG wire#w1
      Contact( "DB611".ParaOut.Out.LoopValves4 )
      Contact( "DB611".ParaOut.Out.EndValve )
   END_RUNG wire#w3
   RUNG wire#w1
      Contact( "DB611".ParaOut.Out.LoopValves5 )
      Contact( "DB611".ParaOut.Out.EndValve )
   END_RUNG wire#w3
   RUNG wire#w1
      Contact( "DB611".ParaOut.Out.LoopValves7 )
      Contact( "DB611".ParaOut.Out.EndValve )
   END_RUNG wire#w3
   RUNG wire#w1
      Contact( "DB611".ParaOut.Out.LoopValves8 )
      Contact( "DB611".ParaOut.Out.EndValve )
   END_RUNG wire#w3
   RUNG wire#w1
      Contact( "DB611".ParaOut.Out.PressureReleaseValves )
   END_RUNG wire#w3
   RUNG wire#w1
      { S7_Templates := "SrcType := Int" } EQ_Contact(in1 := "DB615".CurrentStep, in2 := 2)
      wire#w4
      Contact( "DB609".ParaOut.Out.LoopValves1 )
   END_RUNG wire#w3
   RUNG wire#w1
      { S7_Templates := "SrcType := Int" } EQ_Contact(in1 := "DB615".CurrentStep, in2 := 3)
   END_RUNG wire#w4
   // the same network as SCL:
   "CipVessel".Cv34 := "ModeDb".Cycle4.Selected AND "DB615".CycleRunningMV AND ((("DB615".CurrentStep = 1) AND ("DB604".ParaOut.Out.LoopValves2 OR "DB604".ParaOut.Out.LoopValves3 OR "DB604".ParaOut.Out.LoopValves4 OR "DB604".ParaOut.Out.LoopValves5 OR "DB604".ParaOut.Out.LoopValves7 OR "DB609"."Line Valves")) OR "DB610".ParaOut.Out.LineValves OR ("DB611".ParaOut.Out.LoopValves2 AND "DB611".ParaOut.Out.EndValve) OR ("DB611".ParaOut.Out.LoopValves3 AND "DB611".ParaOut.Out.EndValve) OR ("DB611".ParaOut.Out.LoopValves4 AND "DB611".ParaOut.Out.EndValve) OR ("DB611".ParaOut.Out.LoopValves5 AND "DB611".ParaOut.Out.EndValve) OR ("DB611".ParaOut.Out.LoopValves7 AND "DB611".ParaOut.Out.EndValve) OR ("DB611".ParaOut.Out.LoopValves8 AND "DB611".ParaOut.Out.EndValve) OR "DB611".ParaOut.Out.PressureReleaseValves OR ((("DB615".CurrentStep = 2) OR ("DB615".CurrentStep = 3)) AND "DB609".ParaOut.Out.LoopValves1));
END_REGION

REGION Network 26: ---- REC LINE -------
END_REGION

REGION Network 27: "CipVessel".Cv39
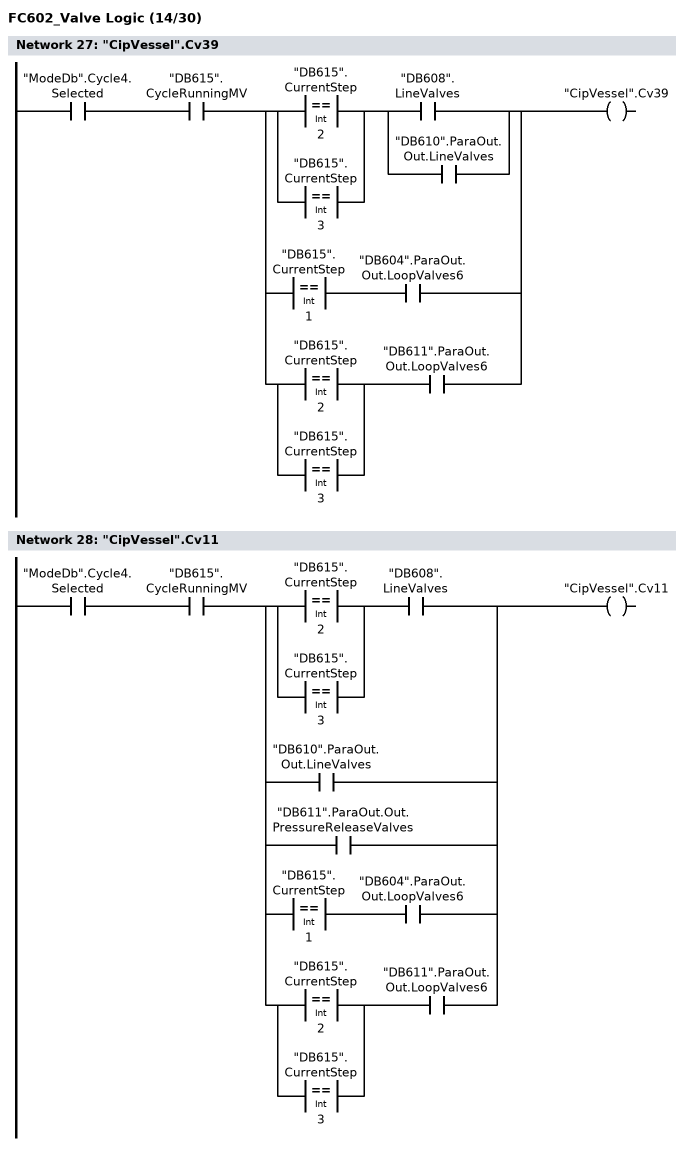
   RUNG wire#powerrail
      Contact( "ModeDb".Cycle4.Selected )
      Contact( "DB615".CycleRunningMV )
      wire#w1
      { S7_Templates := "SrcType := Int" } EQ_Contact(in1 := "DB615".CurrentStep, in2 := 2)
      wire#w2
      Contact( "DB608".LineValves )
      wire#w3
      Coil( "CipVessel".Cv39 )
   END_RUNG
   RUNG wire#w1
      { S7_Templates := "SrcType := Int" } EQ_Contact(in1 := "DB615".CurrentStep, in2 := 3)
   END_RUNG wire#w2
   RUNG wire#w2
      Contact( "DB610".ParaOut.Out.LineValves )
   END_RUNG wire#w3
   RUNG wire#w1
      { S7_Templates := "SrcType := Int" } EQ_Contact(in1 := "DB615".CurrentStep, in2 := 1)
      Contact( "DB604".ParaOut.Out.LoopValves6 )
   END_RUNG wire#w3
   RUNG wire#w1
      { S7_Templates := "SrcType := Int" } EQ_Contact(in1 := "DB615".CurrentStep, in2 := 2)
      wire#w4
      Contact( "DB611".ParaOut.Out.LoopValves6 )
   END_RUNG wire#w3
   RUNG wire#w1
      { S7_Templates := "SrcType := Int" } EQ_Contact(in1 := "DB615".CurrentStep, in2 := 3)
   END_RUNG wire#w4
   // the same network as SCL:
   "CipVessel".Cv39 := "ModeDb".Cycle4.Selected AND "DB615".CycleRunningMV AND (((("DB615".CurrentStep = 2) OR ("DB615".CurrentStep = 3)) AND ("DB608".LineValves OR "DB610".ParaOut.Out.LineValves)) OR (("DB615".CurrentStep = 1) AND "DB604".ParaOut.Out.LoopValves6) OR ((("DB615".CurrentStep = 2) OR ("DB615".CurrentStep = 3)) AND "DB611".ParaOut.Out.LoopValves6));
END_REGION

REGION Network 28: "CipVessel".Cv11
   RUNG wire#powerrail
      Contact( "ModeDb".Cycle4.Selected )
      Contact( "DB615".CycleRunningMV )
      wire#w1
      { S7_Templates := "SrcType := Int" } EQ_Contact(in1 := "DB615".CurrentStep, in2 := 2)
      wire#w2
      Contact( "DB608".LineValves )
      wire#w3
      Coil( "CipVessel".Cv11 )
   END_RUNG
   RUNG wire#w1
      { S7_Templates := "SrcType := Int" } EQ_Contact(in1 := "DB615".CurrentStep, in2 := 3)
   END_RUNG wire#w2
   RUNG wire#w1
      Contact( "DB610".ParaOut.Out.LineValves )
   END_RUNG wire#w3
   RUNG wire#w1
      Contact( "DB611".ParaOut.Out.PressureReleaseValves )
   END_RUNG wire#w3
   RUNG wire#w1
      { S7_Templates := "SrcType := Int" } EQ_Contact(in1 := "DB615".CurrentStep, in2 := 1)
      Contact( "DB604".ParaOut.Out.LoopValves6 )
   END_RUNG wire#w3
   RUNG wire#w1
      { S7_Templates := "SrcType := Int" } EQ_Contact(in1 := "DB615".CurrentStep, in2 := 2)
      wire#w4
      Contact( "DB611".ParaOut.Out.LoopValves6 )
   END_RUNG wire#w3
   RUNG wire#w1
      { S7_Templates := "SrcType := Int" } EQ_Contact(in1 := "DB615".CurrentStep, in2 := 3)
   END_RUNG wire#w4
   // the same network as SCL:
   "CipVessel".Cv11 := "ModeDb".Cycle4.Selected AND "DB615".CycleRunningMV AND (((("DB615".CurrentStep = 2) OR ("DB615".CurrentStep = 3)) AND "DB608".LineValves) OR "DB610".ParaOut.Out.LineValves OR "DB611".ParaOut.Out.PressureReleaseValves OR (("DB615".CurrentStep = 1) AND "DB604".ParaOut.Out.LoopValves6) OR ((("DB615".CurrentStep = 2) OR ("DB615".CurrentStep = 3)) AND "DB611".ParaOut.Out.LoopValves6));
END_REGION

REGION Network 29: -------- PUMP BYPASS LINE ------
END_REGION

REGION Network 30: "CipVessel".Cv31
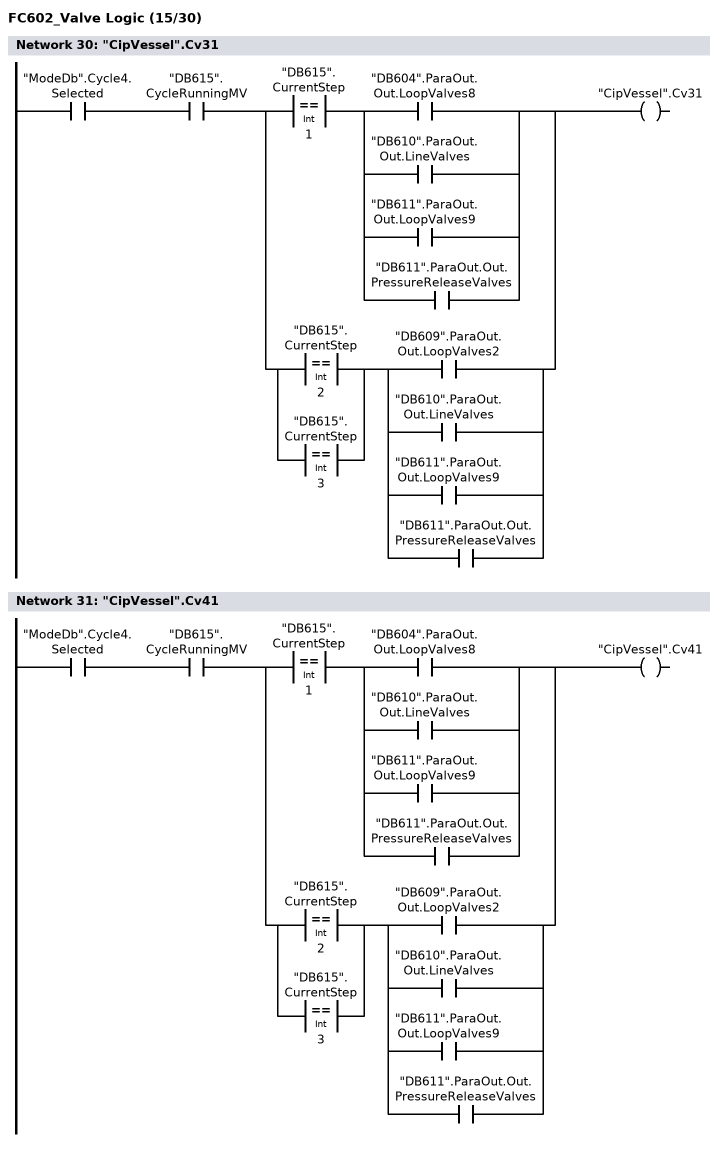
   RUNG wire#powerrail
      Contact( "ModeDb".Cycle4.Selected )
      Contact( "DB615".CycleRunningMV )
      wire#w1
      { S7_Templates := "SrcType := Int" } EQ_Contact(in1 := "DB615".CurrentStep, in2 := 1)
      wire#w2
      Contact( "DB604".ParaOut.Out.LoopValves8 )
      wire#w3
      Coil( "CipVessel".Cv31 )
   END_RUNG
   RUNG wire#w2
      Contact( "DB610".ParaOut.Out.LineValves )
   END_RUNG wire#w3
   RUNG wire#w2
      Contact( "DB611".ParaOut.Out.LoopValves9 )
   END_RUNG wire#w3
   RUNG wire#w2
      Contact( "DB611".ParaOut.Out.PressureReleaseValves )
   END_RUNG wire#w3
   RUNG wire#w1
      { S7_Templates := "SrcType := Int" } EQ_Contact(in1 := "DB615".CurrentStep, in2 := 2)
      wire#w4
      Contact( "DB609".ParaOut.Out.LoopValves2 )
   END_RUNG wire#w3
   RUNG wire#w1
      { S7_Templates := "SrcType := Int" } EQ_Contact(in1 := "DB615".CurrentStep, in2 := 3)
   END_RUNG wire#w4
   RUNG wire#w4
      Contact( "DB610".ParaOut.Out.LineValves )
   END_RUNG wire#w3
   RUNG wire#w4
      Contact( "DB611".ParaOut.Out.LoopValves9 )
   END_RUNG wire#w3
   RUNG wire#w4
      Contact( "DB611".ParaOut.Out.PressureReleaseValves )
   END_RUNG wire#w3
   // the same network as SCL:
   "CipVessel".Cv31 := "ModeDb".Cycle4.Selected AND "DB615".CycleRunningMV AND ((("DB615".CurrentStep = 1) AND ("DB604".ParaOut.Out.LoopValves8 OR "DB610".ParaOut.Out.LineValves OR "DB611".ParaOut.Out.LoopValves9 OR "DB611".ParaOut.Out.PressureReleaseValves)) OR ((("DB615".CurrentStep = 2) OR ("DB615".CurrentStep = 3)) AND ("DB609".ParaOut.Out.LoopValves2 OR "DB610".ParaOut.Out.LineValves OR "DB611".ParaOut.Out.LoopValves9 OR "DB611".ParaOut.Out.PressureReleaseValves)));
END_REGION

REGION Network 31: "CipVessel".Cv41
   RUNG wire#powerrail
      Contact( "ModeDb".Cycle4.Selected )
      Contact( "DB615".CycleRunningMV )
      wire#w1
      { S7_Templates := "SrcType := Int" } EQ_Contact(in1 := "DB615".CurrentStep, in2 := 1)
      wire#w2
      Contact( "DB604".ParaOut.Out.LoopValves8 )
      wire#w3
      Coil( "CipVessel".Cv41 )
   END_RUNG
   RUNG wire#w2
      Contact( "DB610".ParaOut.Out.LineValves )
   END_RUNG wire#w3
   RUNG wire#w2
      Contact( "DB611".ParaOut.Out.LoopValves9 )
   END_RUNG wire#w3
   RUNG wire#w2
      Contact( "DB611".ParaOut.Out.PressureReleaseValves )
   END_RUNG wire#w3
   RUNG wire#w1
      { S7_Templates := "SrcType := Int" } EQ_Contact(in1 := "DB615".CurrentStep, in2 := 2)
      wire#w4
      Contact( "DB609".ParaOut.Out.LoopValves2 )
   END_RUNG wire#w3
   RUNG wire#w1
      { S7_Templates := "SrcType := Int" } EQ_Contact(in1 := "DB615".CurrentStep, in2 := 3)
   END_RUNG wire#w4
   RUNG wire#w4
      Contact( "DB610".ParaOut.Out.LineValves )
   END_RUNG wire#w3
   RUNG wire#w4
      Contact( "DB611".ParaOut.Out.LoopValves9 )
   END_RUNG wire#w3
   RUNG wire#w4
      Contact( "DB611".ParaOut.Out.PressureReleaseValves )
   END_RUNG wire#w3
   // the same network as SCL:
   "CipVessel".Cv41 := "ModeDb".Cycle4.Selected AND "DB615".CycleRunningMV AND ((("DB615".CurrentStep = 1) AND ("DB604".ParaOut.Out.LoopValves8 OR "DB610".ParaOut.Out.LineValves OR "DB611".ParaOut.Out.LoopValves9 OR "DB611".ParaOut.Out.PressureReleaseValves)) OR ((("DB615".CurrentStep = 2) OR ("DB615".CurrentStep = 3)) AND ("DB609".ParaOut.Out.LoopValves2 OR "DB610".ParaOut.Out.LineValves OR "DB611".ParaOut.Out.LoopValves9 OR "DB611".ParaOut.Out.PressureReleaseValves)));
END_REGION

REGION Network 32: -------- PF01 IN LINE ----------
END_REGION

REGION Network 33: "CipVessel".Cv32
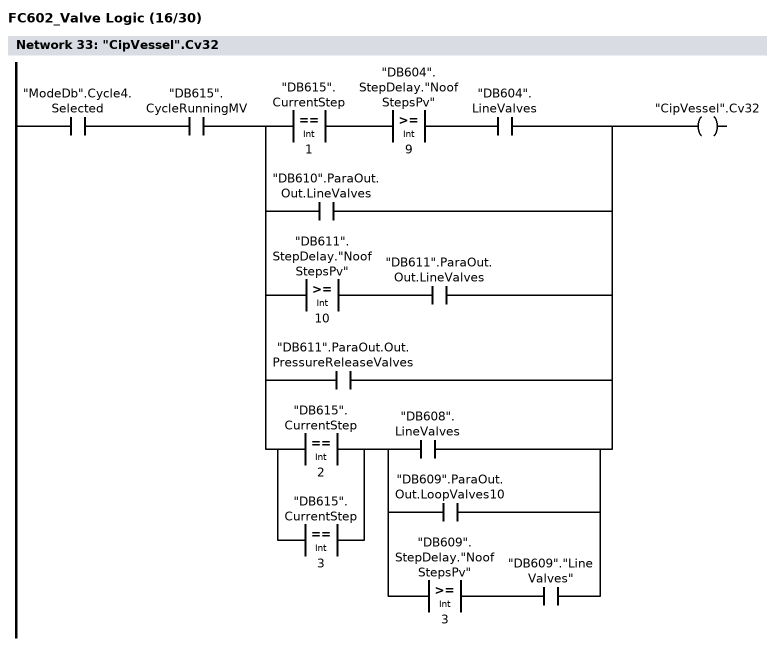
   RUNG wire#powerrail
      Contact( "ModeDb".Cycle4.Selected )
      Contact( "DB615".CycleRunningMV )
      wire#w1
      { S7_Templates := "SrcType := Int" } EQ_Contact(in1 := "DB615".CurrentStep, in2 := 1)
      { S7_Templates := "SrcType := Int" } GE_Contact(in1 := "DB604".StepDelay."Noof StepsPv", in2 := 9)
      Contact( "DB604".LineValves )
      wire#w2
      Coil( "CipVessel".Cv32 )
   END_RUNG
   RUNG wire#w1
      Contact( "DB610".ParaOut.Out.LineValves )
   END_RUNG wire#w2
   RUNG wire#w1
      { S7_Templates := "SrcType := Int" } GE_Contact(in1 := "DB611".StepDelay."Noof StepsPv", in2 := 10)
      Contact( "DB611".ParaOut.Out.LineValves )
   END_RUNG wire#w2
   RUNG wire#w1
      Contact( "DB611".ParaOut.Out.PressureReleaseValves )
   END_RUNG wire#w2
   RUNG wire#w1
      { S7_Templates := "SrcType := Int" } EQ_Contact(in1 := "DB615".CurrentStep, in2 := 2)
      wire#w3
      Contact( "DB608".LineValves )
   END_RUNG wire#w2
   RUNG wire#w1
      { S7_Templates := "SrcType := Int" } EQ_Contact(in1 := "DB615".CurrentStep, in2 := 3)
   END_RUNG wire#w3
   RUNG wire#w3
      Contact( "DB609".ParaOut.Out.LoopValves10 )
   END_RUNG wire#w2
   RUNG wire#w3
      { S7_Templates := "SrcType := Int" } GE_Contact(in1 := "DB609".StepDelay."Noof StepsPv", in2 := 3)
      Contact( "DB609"."Line Valves" )
   END_RUNG wire#w2
   // the same network as SCL:
   "CipVessel".Cv32 := "ModeDb".Cycle4.Selected AND "DB615".CycleRunningMV AND ((("DB615".CurrentStep = 1) AND ("DB604".StepDelay."Noof StepsPv" >= 9) AND "DB604".LineValves) OR "DB610".ParaOut.Out.LineValves OR (("DB611".StepDelay."Noof StepsPv" >= 10) AND "DB611".ParaOut.Out.LineValves) OR "DB611".ParaOut.Out.PressureReleaseValves OR ((("DB615".CurrentStep = 2) OR ("DB615".CurrentStep = 3)) AND ("DB608".LineValves OR "DB609".ParaOut.Out.LoopValves10 OR (("DB609".StepDelay."Noof StepsPv" >= 3) AND "DB609"."Line Valves"))));
END_REGION

REGION Network 34: "CipVessel".Cv40
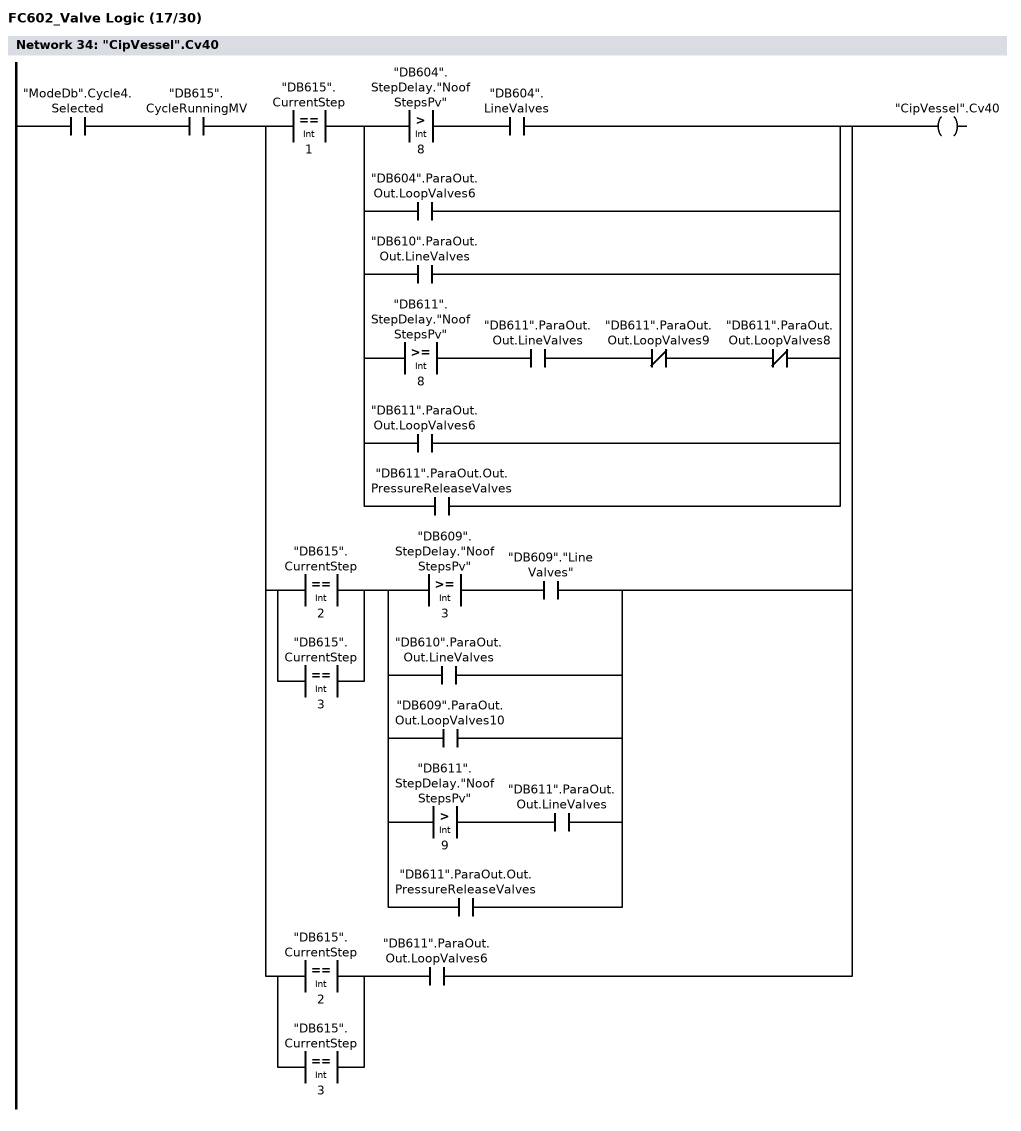
   RUNG wire#powerrail
      Contact( "ModeDb".Cycle4.Selected )
      Contact( "DB615".CycleRunningMV )
      wire#w1
      { S7_Templates := "SrcType := Int" } EQ_Contact(in1 := "DB615".CurrentStep, in2 := 1)
      wire#w2
      { S7_Templates := "SrcType := Int" } GT_Contact(in1 := "DB604".StepDelay."Noof StepsPv", in2 := 8)
      Contact( "DB604".LineValves )
      wire#w3
      Coil( "CipVessel".Cv40 )
   END_RUNG
   RUNG wire#w2
      Contact( "DB604".ParaOut.Out.LoopValves6 )
   END_RUNG wire#w3
   RUNG wire#w2
      Contact( "DB610".ParaOut.Out.LineValves )
   END_RUNG wire#w3
   RUNG wire#w2
      { S7_Templates := "SrcType := Int" } GE_Contact(in1 := "DB611".StepDelay."Noof StepsPv", in2 := 8)
      Contact( "DB611".ParaOut.Out.LineValves )
      I_Contact( "DB611".ParaOut.Out.LoopValves9 )
      I_Contact( "DB611".ParaOut.Out.LoopValves8 )
   END_RUNG wire#w3
   RUNG wire#w2
      Contact( "DB611".ParaOut.Out.LoopValves6 )
   END_RUNG wire#w3
   RUNG wire#w2
      Contact( "DB611".ParaOut.Out.PressureReleaseValves )
   END_RUNG wire#w3
   RUNG wire#w1
      { S7_Templates := "SrcType := Int" } EQ_Contact(in1 := "DB615".CurrentStep, in2 := 2)
      wire#w4
      { S7_Templates := "SrcType := Int" } GE_Contact(in1 := "DB609".StepDelay."Noof StepsPv", in2 := 3)
      Contact( "DB609"."Line Valves" )
   END_RUNG wire#w3
   RUNG wire#w1
      { S7_Templates := "SrcType := Int" } EQ_Contact(in1 := "DB615".CurrentStep, in2 := 3)
   END_RUNG wire#w4
   RUNG wire#w4
      Contact( "DB610".ParaOut.Out.LineValves )
   END_RUNG wire#w3
   RUNG wire#w4
      Contact( "DB609".ParaOut.Out.LoopValves10 )
   END_RUNG wire#w3
   RUNG wire#w4
      { S7_Templates := "SrcType := Int" } GT_Contact(in1 := "DB611".StepDelay."Noof StepsPv", in2 := 9)
      Contact( "DB611".ParaOut.Out.LineValves )
   END_RUNG wire#w3
   RUNG wire#w4
      Contact( "DB611".ParaOut.Out.PressureReleaseValves )
   END_RUNG wire#w3
   RUNG wire#w1
      { S7_Templates := "SrcType := Int" } EQ_Contact(in1 := "DB615".CurrentStep, in2 := 2)
      wire#w5
      Contact( "DB611".ParaOut.Out.LoopValves6 )
   END_RUNG wire#w3
   RUNG wire#w1
      { S7_Templates := "SrcType := Int" } EQ_Contact(in1 := "DB615".CurrentStep, in2 := 3)
   END_RUNG wire#w5
   // the same network as SCL:
   "CipVessel".Cv40 := "ModeDb".Cycle4.Selected AND "DB615".CycleRunningMV AND ((("DB615".CurrentStep = 1) AND ((("DB604".StepDelay."Noof StepsPv" > 8) AND "DB604".LineValves) OR "DB604".ParaOut.Out.LoopValves6 OR "DB610".ParaOut.Out.LineValves OR (("DB611".StepDelay."Noof StepsPv" >= 8) AND "DB611".ParaOut.Out.LineValves AND NOT "DB611".ParaOut.Out.LoopValves9 AND NOT "DB611".ParaOut.Out.LoopValves8) OR "DB611".ParaOut.Out.LoopValves6 OR "DB611".ParaOut.Out.PressureReleaseValves)) OR ((("DB615".CurrentStep = 2) OR ("DB615".CurrentStep = 3)) AND ((("DB609".StepDelay."Noof StepsPv" >= 3) AND "DB609"."Line Valves") OR "DB610".ParaOut.Out.LineValves OR "DB609".ParaOut.Out.LoopValves10 OR (("DB611".StepDelay."Noof StepsPv" > 9) AND "DB611".ParaOut.Out.LineValves) OR "DB611".ParaOut.Out.PressureReleaseValves)) OR ((("DB615".CurrentStep = 2) OR ("DB615".CurrentStep = 3)) AND "DB611".ParaOut.Out.LoopValves6));
END_REGION

REGION Network 35: "CipVessel".Cv44
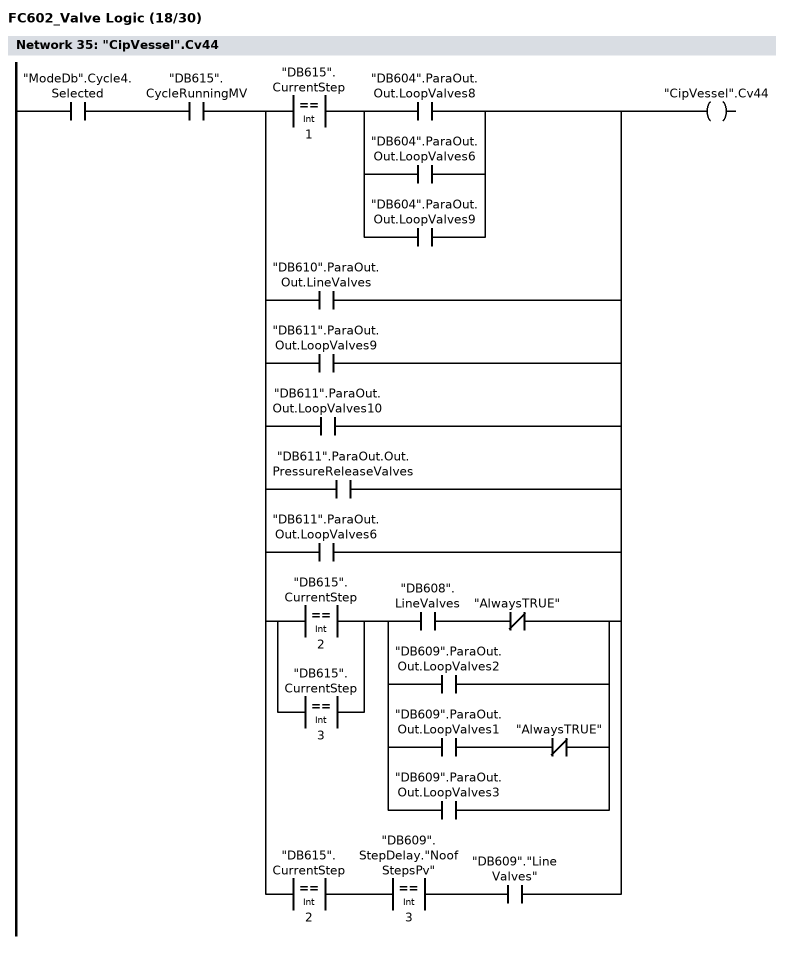
   RUNG wire#powerrail
      Contact( "ModeDb".Cycle4.Selected )
      Contact( "DB615".CycleRunningMV )
      wire#w1
      { S7_Templates := "SrcType := Int" } EQ_Contact(in1 := "DB615".CurrentStep, in2 := 1)
      wire#w2
      Contact( "DB604".ParaOut.Out.LoopValves8 )
      wire#w3
      Coil( "CipVessel".Cv44 )
   END_RUNG
   RUNG wire#w2
      Contact( "DB604".ParaOut.Out.LoopValves6 )
   END_RUNG wire#w3
   RUNG wire#w2
      Contact( "DB604".ParaOut.Out.LoopValves9 )
   END_RUNG wire#w3
   RUNG wire#w1
      Contact( "DB610".ParaOut.Out.LineValves )
   END_RUNG wire#w3
   RUNG wire#w1
      Contact( "DB611".ParaOut.Out.LoopValves9 )
   END_RUNG wire#w3
   RUNG wire#w1
      Contact( "DB611".ParaOut.Out.LoopValves10 )
   END_RUNG wire#w3
   RUNG wire#w1
      Contact( "DB611".ParaOut.Out.PressureReleaseValves )
   END_RUNG wire#w3
   RUNG wire#w1
      Contact( "DB611".ParaOut.Out.LoopValves6 )
   END_RUNG wire#w3
   RUNG wire#w1
      { S7_Templates := "SrcType := Int" } EQ_Contact(in1 := "DB615".CurrentStep, in2 := 2)
      wire#w4
      Contact( "DB608".LineValves )
      I_Contact( "AlwaysTRUE" )
   END_RUNG wire#w3
   RUNG wire#w1
      { S7_Templates := "SrcType := Int" } EQ_Contact(in1 := "DB615".CurrentStep, in2 := 3)
   END_RUNG wire#w4
   RUNG wire#w4
      Contact( "DB609".ParaOut.Out.LoopValves2 )
   END_RUNG wire#w3
   RUNG wire#w4
      Contact( "DB609".ParaOut.Out.LoopValves1 )
      I_Contact( "AlwaysTRUE" )
   END_RUNG wire#w3
   RUNG wire#w4
      Contact( "DB609".ParaOut.Out.LoopValves3 )
   END_RUNG wire#w3
   RUNG wire#w1
      { S7_Templates := "SrcType := Int" } EQ_Contact(in1 := "DB615".CurrentStep, in2 := 2)
      { S7_Templates := "SrcType := Int" } EQ_Contact(in1 := "DB609".StepDelay."Noof StepsPv", in2 := 3)
      Contact( "DB609"."Line Valves" )
   END_RUNG wire#w3
   // the same network as SCL:
   "CipVessel".Cv44 := "ModeDb".Cycle4.Selected AND "DB615".CycleRunningMV AND ((("DB615".CurrentStep = 1) AND ("DB604".ParaOut.Out.LoopValves8 OR "DB604".ParaOut.Out.LoopValves6 OR "DB604".ParaOut.Out.LoopValves9)) OR "DB610".ParaOut.Out.LineValves OR "DB611".ParaOut.Out.LoopValves9 OR "DB611".ParaOut.Out.LoopValves10 OR "DB611".ParaOut.Out.PressureReleaseValves OR "DB611".ParaOut.Out.LoopValves6 OR ((("DB615".CurrentStep = 2) OR ("DB615".CurrentStep = 3)) AND (("DB608".LineValves AND NOT "AlwaysTRUE") OR "DB609".ParaOut.Out.LoopValves2 OR ("DB609".ParaOut.Out.LoopValves1 AND NOT "AlwaysTRUE") OR "DB609".ParaOut.Out.LoopValves3)) OR (("DB615".CurrentStep = 2) AND ("DB609".StepDelay."Noof StepsPv" = 3) AND "DB609"."Line Valves"));
END_REGION

REGION Network 36: "CipVessel".Cv45
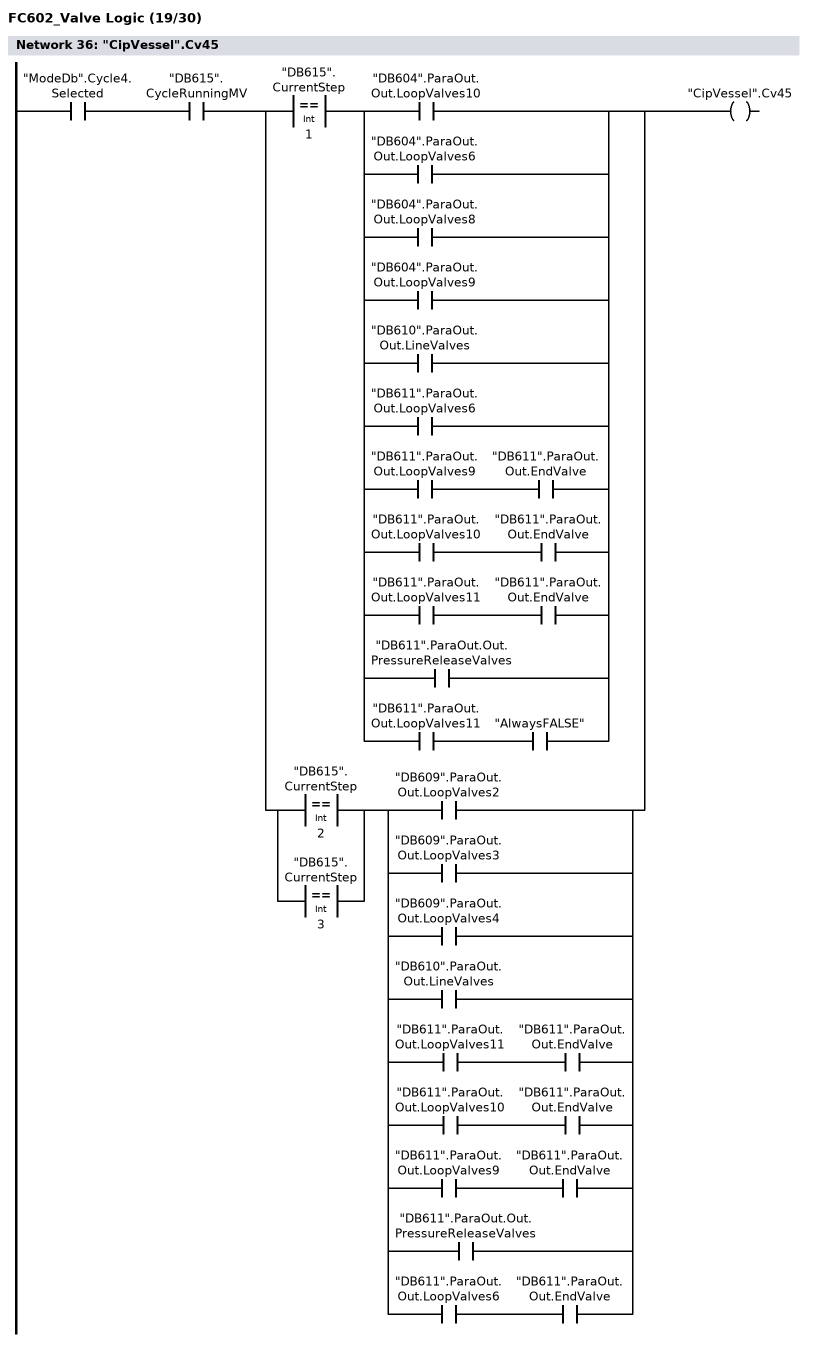
   RUNG wire#powerrail
      Contact( "ModeDb".Cycle4.Selected )
      Contact( "DB615".CycleRunningMV )
      wire#w1
      { S7_Templates := "SrcType := Int" } EQ_Contact(in1 := "DB615".CurrentStep, in2 := 1)
      wire#w2
      Contact( "DB604".ParaOut.Out.LoopValves10 )
      wire#w3
      Coil( "CipVessel".Cv45 )
   END_RUNG
   RUNG wire#w2
      Contact( "DB604".ParaOut.Out.LoopValves6 )
   END_RUNG wire#w3
   RUNG wire#w2
      Contact( "DB604".ParaOut.Out.LoopValves8 )
   END_RUNG wire#w3
   RUNG wire#w2
      Contact( "DB604".ParaOut.Out.LoopValves9 )
   END_RUNG wire#w3
   RUNG wire#w2
      Contact( "DB610".ParaOut.Out.LineValves )
   END_RUNG wire#w3
   RUNG wire#w2
      Contact( "DB611".ParaOut.Out.LoopValves6 )
   END_RUNG wire#w3
   RUNG wire#w2
      Contact( "DB611".ParaOut.Out.LoopValves9 )
      Contact( "DB611".ParaOut.Out.EndValve )
   END_RUNG wire#w3
   RUNG wire#w2
      Contact( "DB611".ParaOut.Out.LoopValves10 )
      Contact( "DB611".ParaOut.Out.EndValve )
   END_RUNG wire#w3
   RUNG wire#w2
      Contact( "DB611".ParaOut.Out.LoopValves11 )
      Contact( "DB611".ParaOut.Out.EndValve )
   END_RUNG wire#w3
   RUNG wire#w2
      Contact( "DB611".ParaOut.Out.PressureReleaseValves )
   END_RUNG wire#w3
   RUNG wire#w2
      Contact( "DB611".ParaOut.Out.LoopValves11 )
      Contact( "AlwaysFALSE" )
   END_RUNG wire#w3
   RUNG wire#w1
      { S7_Templates := "SrcType := Int" } EQ_Contact(in1 := "DB615".CurrentStep, in2 := 2)
      wire#w4
      Contact( "DB609".ParaOut.Out.LoopValves2 )
   END_RUNG wire#w3
   RUNG wire#w1
      { S7_Templates := "SrcType := Int" } EQ_Contact(in1 := "DB615".CurrentStep, in2 := 3)
   END_RUNG wire#w4
   RUNG wire#w4
      Contact( "DB609".ParaOut.Out.LoopValves3 )
   END_RUNG wire#w3
   RUNG wire#w4
      Contact( "DB609".ParaOut.Out.LoopValves4 )
   END_RUNG wire#w3
   RUNG wire#w4
      Contact( "DB610".ParaOut.Out.LineValves )
   END_RUNG wire#w3
   RUNG wire#w4
      Contact( "DB611".ParaOut.Out.LoopValves11 )
      Contact( "DB611".ParaOut.Out.EndValve )
   END_RUNG wire#w3
   RUNG wire#w4
      Contact( "DB611".ParaOut.Out.LoopValves10 )
      Contact( "DB611".ParaOut.Out.EndValve )
   END_RUNG wire#w3
   RUNG wire#w4
      Contact( "DB611".ParaOut.Out.LoopValves9 )
      Contact( "DB611".ParaOut.Out.EndValve )
   END_RUNG wire#w3
   RUNG wire#w4
      Contact( "DB611".ParaOut.Out.PressureReleaseValves )
   END_RUNG wire#w3
   RUNG wire#w4
      Contact( "DB611".ParaOut.Out.LoopValves6 )
      Contact( "DB611".ParaOut.Out.EndValve )
   END_RUNG wire#w3
   // the same network as SCL:
   "CipVessel".Cv45 := "ModeDb".Cycle4.Selected AND "DB615".CycleRunningMV AND ((("DB615".CurrentStep = 1) AND ("DB604".ParaOut.Out.LoopValves10 OR "DB604".ParaOut.Out.LoopValves6 OR "DB604".ParaOut.Out.LoopValves8 OR "DB604".ParaOut.Out.LoopValves9 OR "DB610".ParaOut.Out.LineValves OR "DB611".ParaOut.Out.LoopValves6 OR ("DB611".ParaOut.Out.LoopValves9 AND "DB611".ParaOut.Out.EndValve) OR ("DB611".ParaOut.Out.LoopValves10 AND "DB611".ParaOut.Out.EndValve) OR ("DB611".ParaOut.Out.LoopValves11 AND "DB611".ParaOut.Out.EndValve) OR "DB611".ParaOut.Out.PressureReleaseValves OR ("DB611".ParaOut.Out.LoopValves11 AND "AlwaysFALSE"))) OR ((("DB615".CurrentStep = 2) OR ("DB615".CurrentStep = 3)) AND ("DB609".ParaOut.Out.LoopValves2 OR "DB609".ParaOut.Out.LoopValves3 OR "DB609".ParaOut.Out.LoopValves4 OR "DB610".ParaOut.Out.LineValves OR ("DB611".ParaOut.Out.LoopValves11 AND "DB611".ParaOut.Out.EndValve) OR ("DB611".ParaOut.Out.LoopValves10 AND "DB611".ParaOut.Out.EndValve) OR ("DB611".ParaOut.Out.LoopValves9 AND "DB611".ParaOut.Out.EndValve) OR "DB611".ParaOut.Out.PressureReleaseValves OR ("DB611".ParaOut.Out.LoopValves6 AND "DB611".ParaOut.Out.EndValve))));
END_REGION

REGION Network 37: ----------- PF01 VENT ----------------------
END_REGION

REGION Network 38: "CipVessel".Cv43
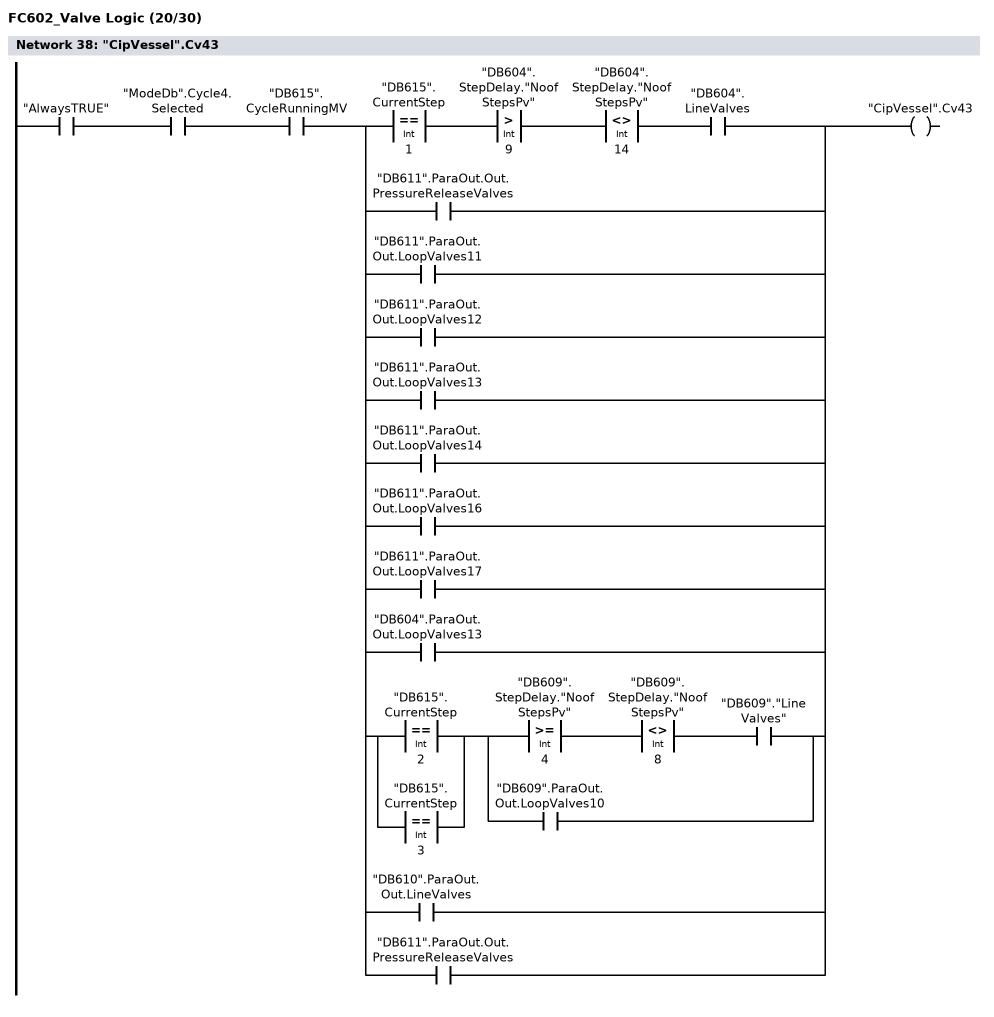
   RUNG wire#powerrail
      Contact( "AlwaysTRUE" )
      Contact( "ModeDb".Cycle4.Selected )
      Contact( "DB615".CycleRunningMV )
      wire#w1
      { S7_Templates := "SrcType := Int" } EQ_Contact(in1 := "DB615".CurrentStep, in2 := 1)
      { S7_Templates := "SrcType := Int" } GT_Contact(in1 := "DB604".StepDelay."Noof StepsPv", in2 := 9)
      { S7_Templates := "SrcType := Int" } NE_Contact(in1 := "DB604".StepDelay."Noof StepsPv", in2 := 14)
      Contact( "DB604".LineValves )
      wire#w2
      Coil( "CipVessel".Cv43 )
   END_RUNG
   RUNG wire#w1
      Contact( "DB611".ParaOut.Out.PressureReleaseValves )
   END_RUNG wire#w2
   RUNG wire#w1
      Contact( "DB611".ParaOut.Out.LoopValves11 )
   END_RUNG wire#w2
   RUNG wire#w1
      Contact( "DB611".ParaOut.Out.LoopValves12 )
   END_RUNG wire#w2
   RUNG wire#w1
      Contact( "DB611".ParaOut.Out.LoopValves13 )
   END_RUNG wire#w2
   RUNG wire#w1
      Contact( "DB611".ParaOut.Out.LoopValves14 )
   END_RUNG wire#w2
   RUNG wire#w1
      Contact( "DB611".ParaOut.Out.LoopValves16 )
   END_RUNG wire#w2
   RUNG wire#w1
      Contact( "DB611".ParaOut.Out.LoopValves17 )
   END_RUNG wire#w2
   RUNG wire#w1
      Contact( "DB604".ParaOut.Out.LoopValves13 )
   END_RUNG wire#w2
   RUNG wire#w1
      { S7_Templates := "SrcType := Int" } EQ_Contact(in1 := "DB615".CurrentStep, in2 := 2)
      wire#w3
      { S7_Templates := "SrcType := Int" } GE_Contact(in1 := "DB609".StepDelay."Noof StepsPv", in2 := 4)
      { S7_Templates := "SrcType := Int" } NE_Contact(in1 := "DB609".StepDelay."Noof StepsPv", in2 := 8)
      Contact( "DB609"."Line Valves" )
   END_RUNG wire#w2
   RUNG wire#w1
      { S7_Templates := "SrcType := Int" } EQ_Contact(in1 := "DB615".CurrentStep, in2 := 3)
   END_RUNG wire#w3
   RUNG wire#w3
      Contact( "DB609".ParaOut.Out.LoopValves10 )
   END_RUNG wire#w2
   RUNG wire#w1
      Contact( "DB610".ParaOut.Out.LineValves )
   END_RUNG wire#w2
   RUNG wire#w1
      Contact( "DB611".ParaOut.Out.PressureReleaseValves )
   END_RUNG wire#w2
   // the same network as SCL:
   "CipVessel".Cv43 := "AlwaysTRUE" AND "ModeDb".Cycle4.Selected AND "DB615".CycleRunningMV AND ((("DB615".CurrentStep = 1) AND ("DB604".StepDelay."Noof StepsPv" > 9) AND ("DB604".StepDelay."Noof StepsPv" <> 14) AND "DB604".LineValves) OR "DB611".ParaOut.Out.PressureReleaseValves OR "DB611".ParaOut.Out.LoopValves11 OR "DB611".ParaOut.Out.LoopValves12 OR "DB611".ParaOut.Out.LoopValves13 OR "DB611".ParaOut.Out.LoopValves14 OR "DB611".ParaOut.Out.LoopValves16 OR "DB611".ParaOut.Out.LoopValves17 OR "DB604".ParaOut.Out.LoopValves13 OR ((("DB615".CurrentStep = 2) OR ("DB615".CurrentStep = 3)) AND ((("DB609".StepDelay."Noof StepsPv" >= 4) AND ("DB609".StepDelay."Noof StepsPv" <> 8) AND "DB609"."Line Valves") OR "DB609".ParaOut.Out.LoopValves10)) OR "DB610".ParaOut.Out.LineValves OR "DB611".ParaOut.Out.PressureReleaseValves);
END_REGION

REGION Network 39: "CipVessel".Cv47
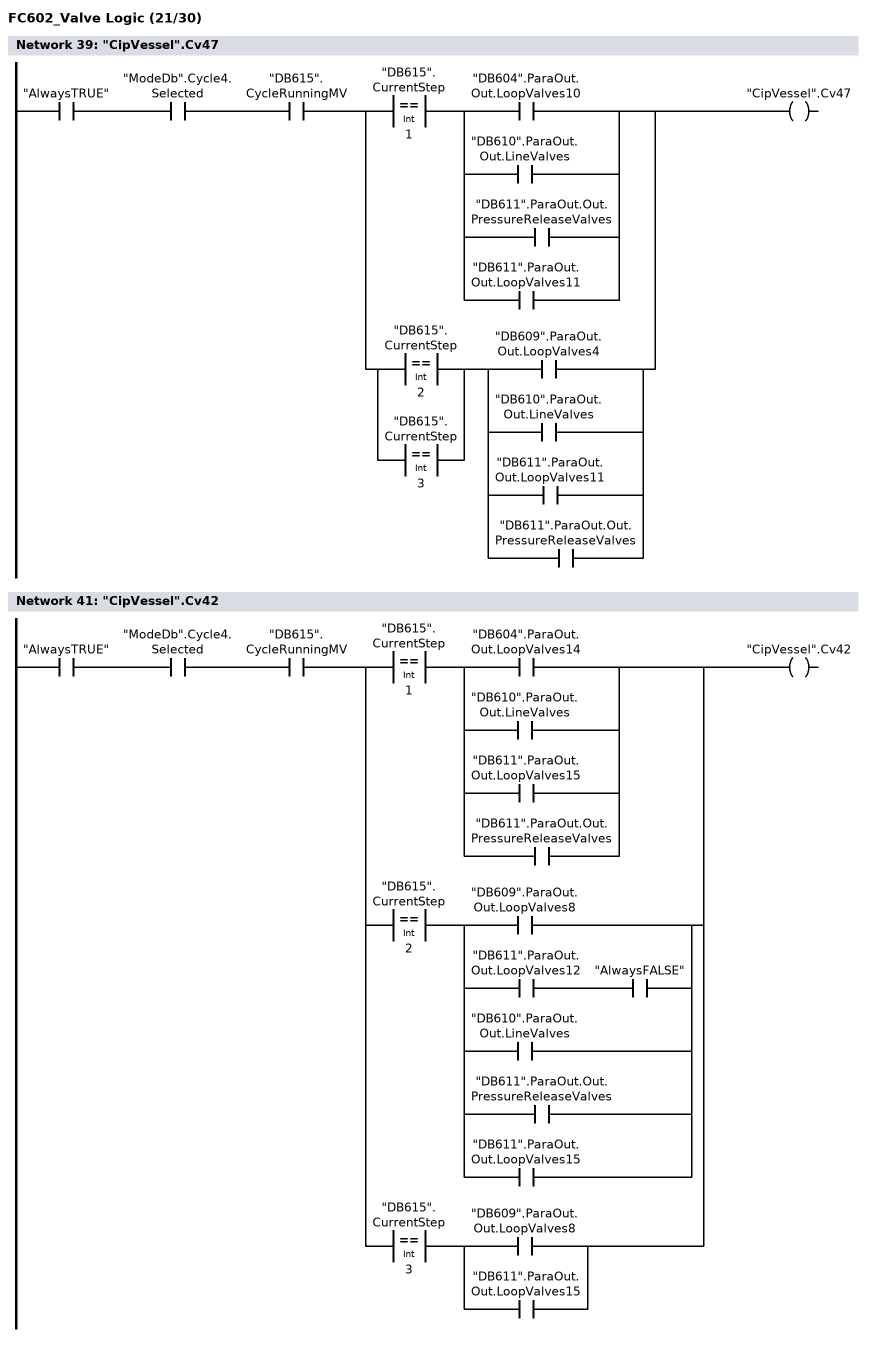
   RUNG wire#powerrail
      Contact( "AlwaysTRUE" )
      Contact( "ModeDb".Cycle4.Selected )
      Contact( "DB615".CycleRunningMV )
      wire#w1
      { S7_Templates := "SrcType := Int" } EQ_Contact(in1 := "DB615".CurrentStep, in2 := 1)
      wire#w2
      Contact( "DB604".ParaOut.Out.LoopValves10 )
      wire#w3
      Coil( "CipVessel".Cv47 )
   END_RUNG
   RUNG wire#w2
      Contact( "DB610".ParaOut.Out.LineValves )
   END_RUNG wire#w3
   RUNG wire#w2
      Contact( "DB611".ParaOut.Out.PressureReleaseValves )
   END_RUNG wire#w3
   RUNG wire#w2
      Contact( "DB611".ParaOut.Out.LoopValves11 )
   END_RUNG wire#w3
   RUNG wire#w1
      { S7_Templates := "SrcType := Int" } EQ_Contact(in1 := "DB615".CurrentStep, in2 := 2)
      wire#w4
      Contact( "DB609".ParaOut.Out.LoopValves4 )
   END_RUNG wire#w3
   RUNG wire#w1
      { S7_Templates := "SrcType := Int" } EQ_Contact(in1 := "DB615".CurrentStep, in2 := 3)
   END_RUNG wire#w4
   RUNG wire#w4
      Contact( "DB610".ParaOut.Out.LineValves )
   END_RUNG wire#w3
   RUNG wire#w4
      Contact( "DB611".ParaOut.Out.LoopValves11 )
   END_RUNG wire#w3
   RUNG wire#w4
      Contact( "DB611".ParaOut.Out.PressureReleaseValves )
   END_RUNG wire#w3
   // the same network as SCL:
   "CipVessel".Cv47 := "AlwaysTRUE" AND "ModeDb".Cycle4.Selected AND "DB615".CycleRunningMV AND ((("DB615".CurrentStep = 1) AND ("DB604".ParaOut.Out.LoopValves10 OR "DB610".ParaOut.Out.LineValves OR "DB611".ParaOut.Out.PressureReleaseValves OR "DB611".ParaOut.Out.LoopValves11)) OR ((("DB615".CurrentStep = 2) OR ("DB615".CurrentStep = 3)) AND ("DB609".ParaOut.Out.LoopValves4 OR "DB610".ParaOut.Out.LineValves OR "DB611".ParaOut.Out.LoopValves11 OR "DB611".ParaOut.Out.PressureReleaseValves)));
END_REGION

REGION Network 40: -------- PF01 BYPASS LINE ----
END_REGION

REGION Network 41: "CipVessel".Cv42
   RUNG wire#powerrail
      Contact( "AlwaysTRUE" )
      Contact( "ModeDb".Cycle4.Selected )
      Contact( "DB615".CycleRunningMV )
      wire#w1
      { S7_Templates := "SrcType := Int" } EQ_Contact(in1 := "DB615".CurrentStep, in2 := 1)
      wire#w2
      Contact( "DB604".ParaOut.Out.LoopValves14 )
      wire#w3
      Coil( "CipVessel".Cv42 )
   END_RUNG
   RUNG wire#w2
      Contact( "DB610".ParaOut.Out.LineValves )
   END_RUNG wire#w3
   RUNG wire#w2
      Contact( "DB611".ParaOut.Out.LoopValves15 )
   END_RUNG wire#w3
   RUNG wire#w2
      Contact( "DB611".ParaOut.Out.PressureReleaseValves )
   END_RUNG wire#w3
   RUNG wire#w1
      { S7_Templates := "SrcType := Int" } EQ_Contact(in1 := "DB615".CurrentStep, in2 := 2)
      wire#w4
      Contact( "DB609".ParaOut.Out.LoopValves8 )
   END_RUNG wire#w3
   RUNG wire#w4
      Contact( "DB611".ParaOut.Out.LoopValves12 )
      Contact( "AlwaysFALSE" )
   END_RUNG wire#w3
   RUNG wire#w4
      Contact( "DB610".ParaOut.Out.LineValves )
   END_RUNG wire#w3
   RUNG wire#w4
      Contact( "DB611".ParaOut.Out.PressureReleaseValves )
   END_RUNG wire#w3
   RUNG wire#w4
      Contact( "DB611".ParaOut.Out.LoopValves15 )
   END_RUNG wire#w3
   RUNG wire#w1
      { S7_Templates := "SrcType := Int" } EQ_Contact(in1 := "DB615".CurrentStep, in2 := 3)
      wire#w5
      Contact( "DB609".ParaOut.Out.LoopValves8 )
   END_RUNG wire#w3
   RUNG wire#w5
      Contact( "DB611".ParaOut.Out.LoopValves15 )
   END_RUNG wire#w3
   // the same network as SCL:
   "CipVessel".Cv42 := "AlwaysTRUE" AND "ModeDb".Cycle4.Selected AND "DB615".CycleRunningMV AND ((("DB615".CurrentStep = 1) AND ("DB604".ParaOut.Out.LoopValves14 OR "DB610".ParaOut.Out.LineValves OR "DB611".ParaOut.Out.LoopValves15 OR "DB611".ParaOut.Out.PressureReleaseValves)) OR (("DB615".CurrentStep = 2) AND ("DB609".ParaOut.Out.LoopValves8 OR ("DB611".ParaOut.Out.LoopValves12 AND "AlwaysFALSE") OR "DB610".ParaOut.Out.LineValves OR "DB611".ParaOut.Out.PressureReleaseValves OR "DB611".ParaOut.Out.LoopValves15)) OR (("DB615".CurrentStep = 3) AND ("DB609".ParaOut.Out.LoopValves8 OR "DB611".ParaOut.Out.LoopValves15)));
END_REGION

REGION Network 42: "CipVessel".Cv48
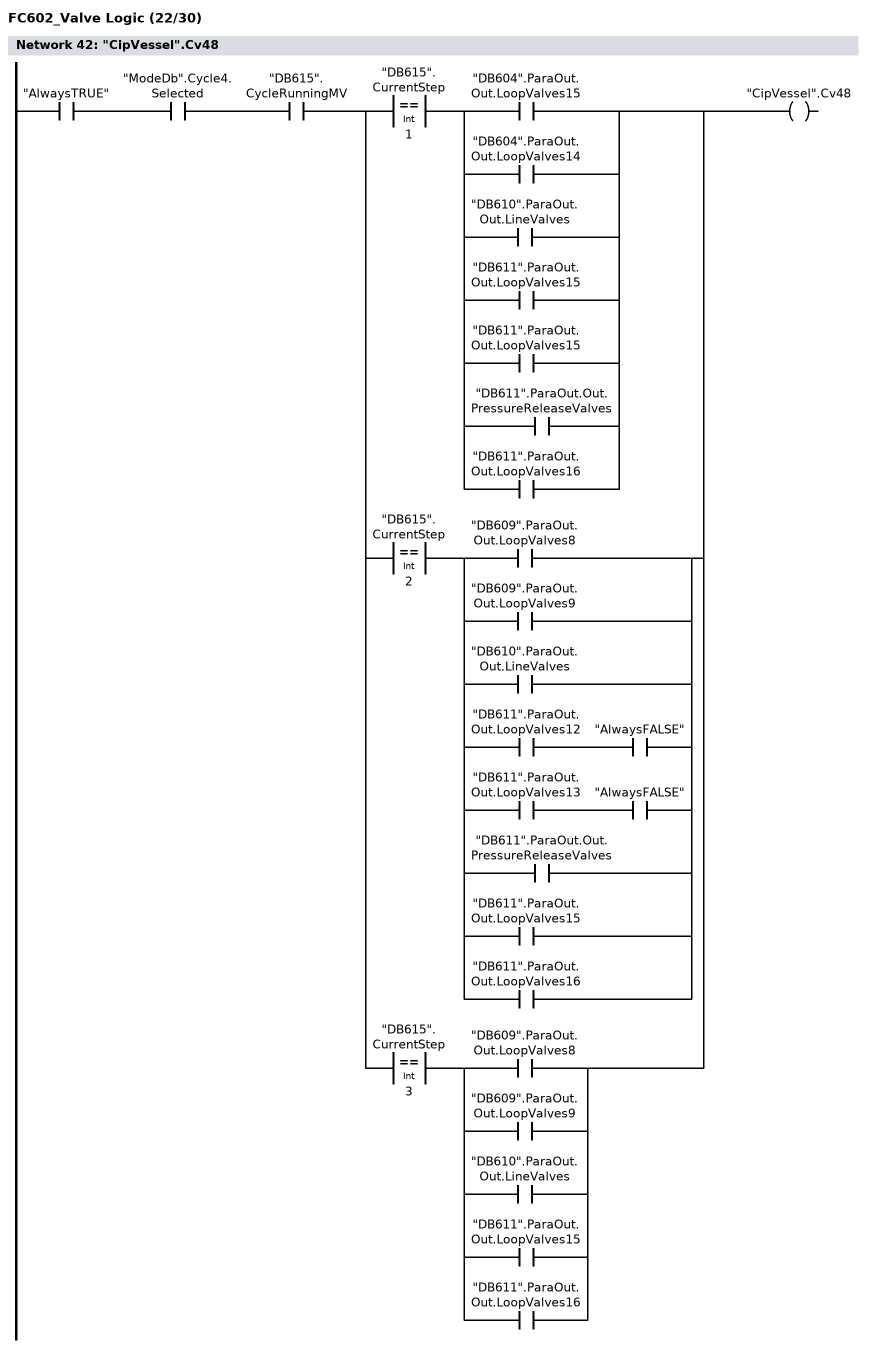
   RUNG wire#powerrail
      Contact( "AlwaysTRUE" )
      Contact( "ModeDb".Cycle4.Selected )
      Contact( "DB615".CycleRunningMV )
      wire#w1
      { S7_Templates := "SrcType := Int" } EQ_Contact(in1 := "DB615".CurrentStep, in2 := 1)
      wire#w2
      Contact( "DB604".ParaOut.Out.LoopValves15 )
      wire#w3
      Coil( "CipVessel".Cv48 )
   END_RUNG
   RUNG wire#w2
      Contact( "DB604".ParaOut.Out.LoopValves14 )
   END_RUNG wire#w3
   RUNG wire#w2
      Contact( "DB610".ParaOut.Out.LineValves )
   END_RUNG wire#w3
   RUNG wire#w2
      Contact( "DB611".ParaOut.Out.LoopValves15 )
   END_RUNG wire#w3
   RUNG wire#w2
      Contact( "DB611".ParaOut.Out.LoopValves15 )
   END_RUNG wire#w3
   RUNG wire#w2
      Contact( "DB611".ParaOut.Out.PressureReleaseValves )
   END_RUNG wire#w3
   RUNG wire#w2
      Contact( "DB611".ParaOut.Out.LoopValves16 )
   END_RUNG wire#w3
   RUNG wire#w1
      { S7_Templates := "SrcType := Int" } EQ_Contact(in1 := "DB615".CurrentStep, in2 := 2)
      wire#w4
      Contact( "DB609".ParaOut.Out.LoopValves8 )
   END_RUNG wire#w3
   RUNG wire#w4
      Contact( "DB609".ParaOut.Out.LoopValves9 )
   END_RUNG wire#w3
   RUNG wire#w4
      Contact( "DB610".ParaOut.Out.LineValves )
   END_RUNG wire#w3
   RUNG wire#w4
      Contact( "DB611".ParaOut.Out.LoopValves12 )
      Contact( "AlwaysFALSE" )
   END_RUNG wire#w3
   RUNG wire#w4
      Contact( "DB611".ParaOut.Out.LoopValves13 )
      Contact( "AlwaysFALSE" )
   END_RUNG wire#w3
   RUNG wire#w4
      Contact( "DB611".ParaOut.Out.PressureReleaseValves )
   END_RUNG wire#w3
   RUNG wire#w4
      Contact( "DB611".ParaOut.Out.LoopValves15 )
   END_RUNG wire#w3
   RUNG wire#w4
      Contact( "DB611".ParaOut.Out.LoopValves16 )
   END_RUNG wire#w3
   RUNG wire#w1
      { S7_Templates := "SrcType := Int" } EQ_Contact(in1 := "DB615".CurrentStep, in2 := 3)
      wire#w5
      Contact( "DB609".ParaOut.Out.LoopValves8 )
   END_RUNG wire#w3
   RUNG wire#w5
      Contact( "DB609".ParaOut.Out.LoopValves9 )
   END_RUNG wire#w3
   RUNG wire#w5
      Contact( "DB610".ParaOut.Out.LineValves )
   END_RUNG wire#w3
   RUNG wire#w5
      Contact( "DB611".ParaOut.Out.LoopValves15 )
   END_RUNG wire#w3
   RUNG wire#w5
      Contact( "DB611".ParaOut.Out.LoopValves16 )
   END_RUNG wire#w3
   // the same network as SCL:
   "CipVessel".Cv48 := "AlwaysTRUE" AND "ModeDb".Cycle4.Selected AND "DB615".CycleRunningMV AND ((("DB615".CurrentStep = 1) AND ("DB604".ParaOut.Out.LoopValves15 OR "DB604".ParaOut.Out.LoopValves14 OR "DB610".ParaOut.Out.LineValves OR "DB611".ParaOut.Out.LoopValves15 OR "DB611".ParaOut.Out.LoopValves15 OR "DB611".ParaOut.Out.PressureReleaseValves OR "DB611".ParaOut.Out.LoopValves16)) OR (("DB615".CurrentStep = 2) AND ("DB609".ParaOut.Out.LoopValves8 OR "DB609".ParaOut.Out.LoopValves9 OR "DB610".ParaOut.Out.LineValves OR ("DB611".ParaOut.Out.LoopValves12 AND "AlwaysFALSE") OR ("DB611".ParaOut.Out.LoopValves13 AND "AlwaysFALSE") OR "DB611".ParaOut.Out.PressureReleaseValves OR "DB611".ParaOut.Out.LoopValves15 OR "DB611".ParaOut.Out.LoopValves16)) OR (("DB615".CurrentStep = 3) AND ("DB609".ParaOut.Out.LoopValves8 OR "DB609".ParaOut.Out.LoopValves9 OR "DB610".ParaOut.Out.LineValves OR "DB611".ParaOut.Out.LoopValves15 OR "DB611".ParaOut.Out.LoopValves16)));
END_REGION

REGION Network 43: ---------- PF02 IN LINE --------
END_REGION

REGION Network 44: "CipVessel".Cv50
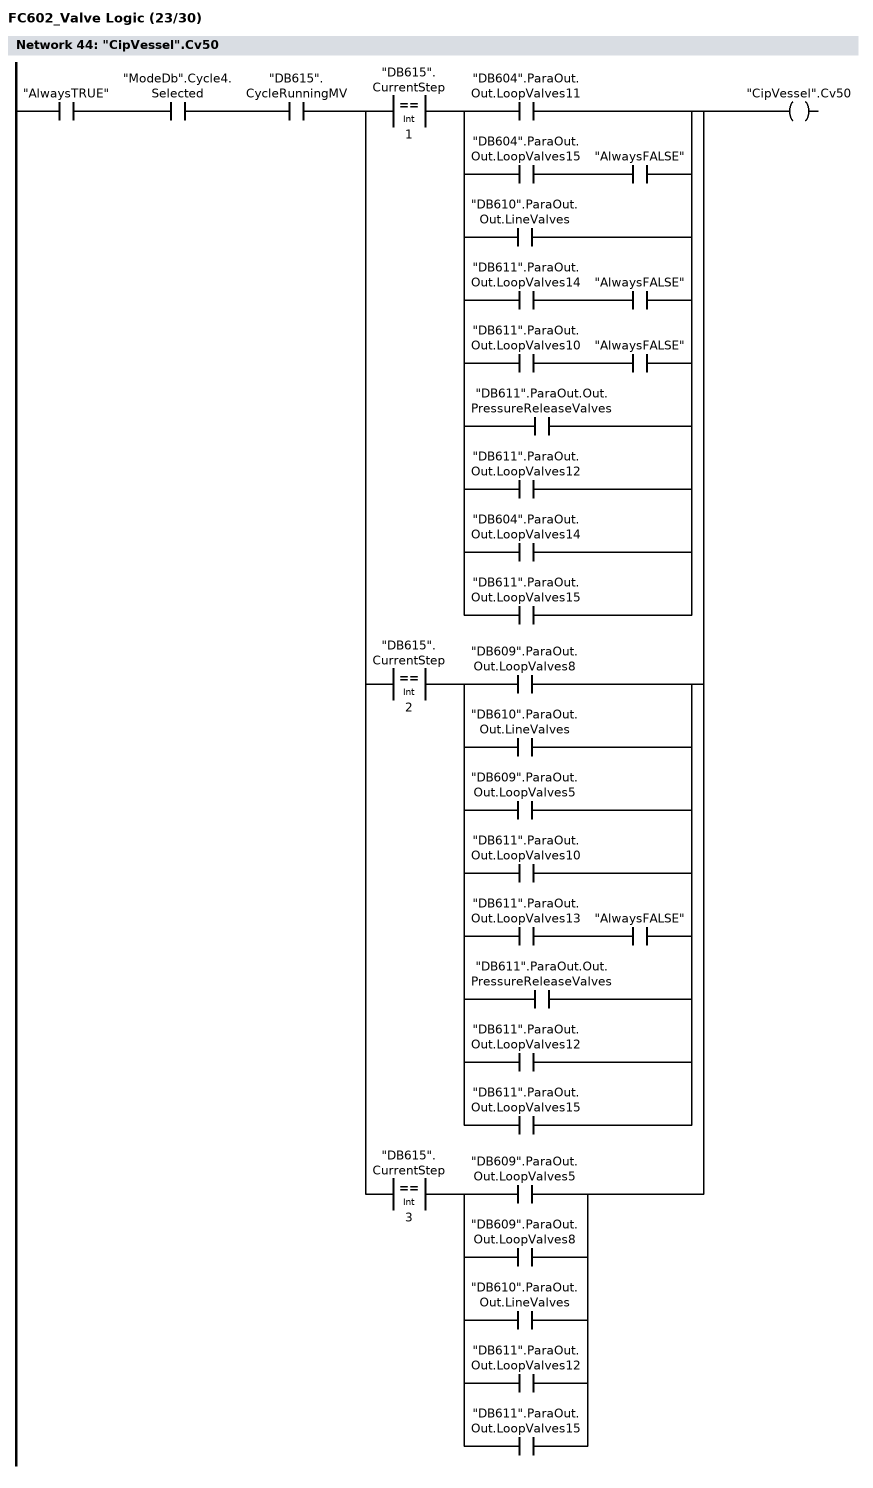
   RUNG wire#powerrail
      Contact( "AlwaysTRUE" )
      Contact( "ModeDb".Cycle4.Selected )
      Contact( "DB615".CycleRunningMV )
      wire#w1
      { S7_Templates := "SrcType := Int" } EQ_Contact(in1 := "DB615".CurrentStep, in2 := 1)
      wire#w2
      Contact( "DB604".ParaOut.Out.LoopValves11 )
      wire#w3
      Coil( "CipVessel".Cv50 )
   END_RUNG
   RUNG wire#w2
      Contact( "DB604".ParaOut.Out.LoopValves15 )
      Contact( "AlwaysFALSE" )
   END_RUNG wire#w3
   RUNG wire#w2
      Contact( "DB610".ParaOut.Out.LineValves )
   END_RUNG wire#w3
   RUNG wire#w2
      Contact( "DB611".ParaOut.Out.LoopValves14 )
      Contact( "AlwaysFALSE" )
   END_RUNG wire#w3
   RUNG wire#w2
      Contact( "DB611".ParaOut.Out.LoopValves10 )
      Contact( "AlwaysFALSE" )
   END_RUNG wire#w3
   RUNG wire#w2
      Contact( "DB611".ParaOut.Out.PressureReleaseValves )
   END_RUNG wire#w3
   RUNG wire#w2
      Contact( "DB611".ParaOut.Out.LoopValves12 )
   END_RUNG wire#w3
   RUNG wire#w2
      Contact( "DB604".ParaOut.Out.LoopValves14 )
   END_RUNG wire#w3
   RUNG wire#w2
      Contact( "DB611".ParaOut.Out.LoopValves15 )
   END_RUNG wire#w3
   RUNG wire#w1
      { S7_Templates := "SrcType := Int" } EQ_Contact(in1 := "DB615".CurrentStep, in2 := 2)
      wire#w4
      Contact( "DB609".ParaOut.Out.LoopValves8 )
   END_RUNG wire#w3
   RUNG wire#w4
      Contact( "DB610".ParaOut.Out.LineValves )
   END_RUNG wire#w3
   RUNG wire#w4
      Contact( "DB609".ParaOut.Out.LoopValves5 )
   END_RUNG wire#w3
   RUNG wire#w4
      Contact( "DB611".ParaOut.Out.LoopValves10 )
   END_RUNG wire#w3
   RUNG wire#w4
      Contact( "DB611".ParaOut.Out.LoopValves13 )
      Contact( "AlwaysFALSE" )
   END_RUNG wire#w3
   RUNG wire#w4
      Contact( "DB611".ParaOut.Out.PressureReleaseValves )
   END_RUNG wire#w3
   RUNG wire#w4
      Contact( "DB611".ParaOut.Out.LoopValves12 )
   END_RUNG wire#w3
   RUNG wire#w4
      Contact( "DB611".ParaOut.Out.LoopValves15 )
   END_RUNG wire#w3
   RUNG wire#w1
      { S7_Templates := "SrcType := Int" } EQ_Contact(in1 := "DB615".CurrentStep, in2 := 3)
      wire#w5
      Contact( "DB609".ParaOut.Out.LoopValves5 )
   END_RUNG wire#w3
   RUNG wire#w5
      Contact( "DB609".ParaOut.Out.LoopValves8 )
   END_RUNG wire#w3
   RUNG wire#w5
      Contact( "DB610".ParaOut.Out.LineValves )
   END_RUNG wire#w3
   RUNG wire#w5
      Contact( "DB611".ParaOut.Out.LoopValves12 )
   END_RUNG wire#w3
   RUNG wire#w5
      Contact( "DB611".ParaOut.Out.LoopValves15 )
   END_RUNG wire#w3
   // the same network as SCL:
   "CipVessel".Cv50 := "AlwaysTRUE" AND "ModeDb".Cycle4.Selected AND "DB615".CycleRunningMV AND ((("DB615".CurrentStep = 1) AND ("DB604".ParaOut.Out.LoopValves11 OR ("DB604".ParaOut.Out.LoopValves15 AND "AlwaysFALSE") OR "DB610".ParaOut.Out.LineValves OR ("DB611".ParaOut.Out.LoopValves14 AND "AlwaysFALSE") OR ("DB611".ParaOut.Out.LoopValves10 AND "AlwaysFALSE") OR "DB611".ParaOut.Out.PressureReleaseValves OR "DB611".ParaOut.Out.LoopValves12 OR "DB604".ParaOut.Out.LoopValves14 OR "DB611".ParaOut.Out.LoopValves15)) OR (("DB615".CurrentStep = 2) AND ("DB609".ParaOut.Out.LoopValves8 OR "DB610".ParaOut.Out.LineValves OR "DB609".ParaOut.Out.LoopValves5 OR "DB611".ParaOut.Out.LoopValves10 OR ("DB611".ParaOut.Out.LoopValves13 AND "AlwaysFALSE") OR "DB611".ParaOut.Out.PressureReleaseValves OR "DB611".ParaOut.Out.LoopValves12 OR "DB611".ParaOut.Out.LoopValves15)) OR (("DB615".CurrentStep = 3) AND ("DB609".ParaOut.Out.LoopValves5 OR "DB609".ParaOut.Out.LoopValves8 OR "DB610".ParaOut.Out.LineValves OR "DB611".ParaOut.Out.LoopValves12 OR "DB611".ParaOut.Out.LoopValves15)));
END_REGION

REGION Network 45: "CipVessel".Cv51
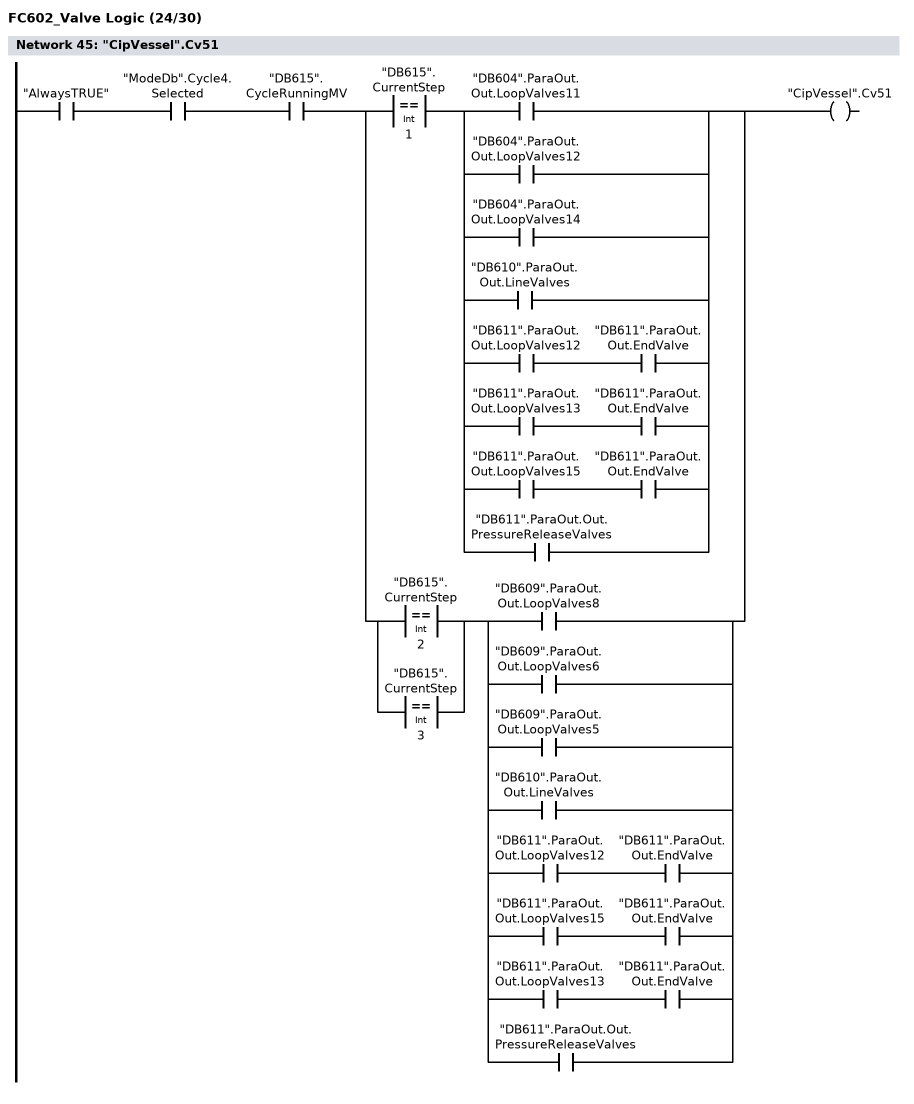
   RUNG wire#powerrail
      Contact( "AlwaysTRUE" )
      Contact( "ModeDb".Cycle4.Selected )
      Contact( "DB615".CycleRunningMV )
      wire#w1
      { S7_Templates := "SrcType := Int" } EQ_Contact(in1 := "DB615".CurrentStep, in2 := 1)
      wire#w2
      Contact( "DB604".ParaOut.Out.LoopValves11 )
      wire#w3
      Coil( "CipVessel".Cv51 )
   END_RUNG
   RUNG wire#w2
      Contact( "DB604".ParaOut.Out.LoopValves12 )
   END_RUNG wire#w3
   RUNG wire#w2
      Contact( "DB604".ParaOut.Out.LoopValves14 )
   END_RUNG wire#w3
   RUNG wire#w2
      Contact( "DB610".ParaOut.Out.LineValves )
   END_RUNG wire#w3
   RUNG wire#w2
      Contact( "DB611".ParaOut.Out.LoopValves12 )
      Contact( "DB611".ParaOut.Out.EndValve )
   END_RUNG wire#w3
   RUNG wire#w2
      Contact( "DB611".ParaOut.Out.LoopValves13 )
      Contact( "DB611".ParaOut.Out.EndValve )
   END_RUNG wire#w3
   RUNG wire#w2
      Contact( "DB611".ParaOut.Out.LoopValves15 )
      Contact( "DB611".ParaOut.Out.EndValve )
   END_RUNG wire#w3
   RUNG wire#w2
      Contact( "DB611".ParaOut.Out.PressureReleaseValves )
   END_RUNG wire#w3
   RUNG wire#w1
      { S7_Templates := "SrcType := Int" } EQ_Contact(in1 := "DB615".CurrentStep, in2 := 2)
      wire#w4
      Contact( "DB609".ParaOut.Out.LoopValves8 )
   END_RUNG wire#w3
   RUNG wire#w1
      { S7_Templates := "SrcType := Int" } EQ_Contact(in1 := "DB615".CurrentStep, in2 := 3)
   END_RUNG wire#w4
   RUNG wire#w4
      Contact( "DB609".ParaOut.Out.LoopValves6 )
   END_RUNG wire#w3
   RUNG wire#w4
      Contact( "DB609".ParaOut.Out.LoopValves5 )
   END_RUNG wire#w3
   RUNG wire#w4
      Contact( "DB610".ParaOut.Out.LineValves )
   END_RUNG wire#w3
   RUNG wire#w4
      Contact( "DB611".ParaOut.Out.LoopValves12 )
      Contact( "DB611".ParaOut.Out.EndValve )
   END_RUNG wire#w3
   RUNG wire#w4
      Contact( "DB611".ParaOut.Out.LoopValves15 )
      Contact( "DB611".ParaOut.Out.EndValve )
   END_RUNG wire#w3
   RUNG wire#w4
      Contact( "DB611".ParaOut.Out.LoopValves13 )
      Contact( "DB611".ParaOut.Out.EndValve )
   END_RUNG wire#w3
   RUNG wire#w4
      Contact( "DB611".ParaOut.Out.PressureReleaseValves )
   END_RUNG wire#w3
   // the same network as SCL:
   "CipVessel".Cv51 := "AlwaysTRUE" AND "ModeDb".Cycle4.Selected AND "DB615".CycleRunningMV AND ((("DB615".CurrentStep = 1) AND ("DB604".ParaOut.Out.LoopValves11 OR "DB604".ParaOut.Out.LoopValves12 OR "DB604".ParaOut.Out.LoopValves14 OR "DB610".ParaOut.Out.LineValves OR ("DB611".ParaOut.Out.LoopValves12 AND "DB611".ParaOut.Out.EndValve) OR ("DB611".ParaOut.Out.LoopValves13 AND "DB611".ParaOut.Out.EndValve) OR ("DB611".ParaOut.Out.LoopValves15 AND "DB611".ParaOut.Out.EndValve) OR "DB611".ParaOut.Out.PressureReleaseValves)) OR ((("DB615".CurrentStep = 2) OR ("DB615".CurrentStep = 3)) AND ("DB609".ParaOut.Out.LoopValves8 OR "DB609".ParaOut.Out.LoopValves6 OR "DB609".ParaOut.Out.LoopValves5 OR "DB610".ParaOut.Out.LineValves OR ("DB611".ParaOut.Out.LoopValves12 AND "DB611".ParaOut.Out.EndValve) OR ("DB611".ParaOut.Out.LoopValves15 AND "DB611".ParaOut.Out.EndValve) OR ("DB611".ParaOut.Out.LoopValves13 AND "DB611".ParaOut.Out.EndValve) OR "DB611".ParaOut.Out.PressureReleaseValves)));
END_REGION

REGION Network 46: ----------- PF02 VENT -------------
END_REGION

REGION Network 47: "CipVessel".Cv49
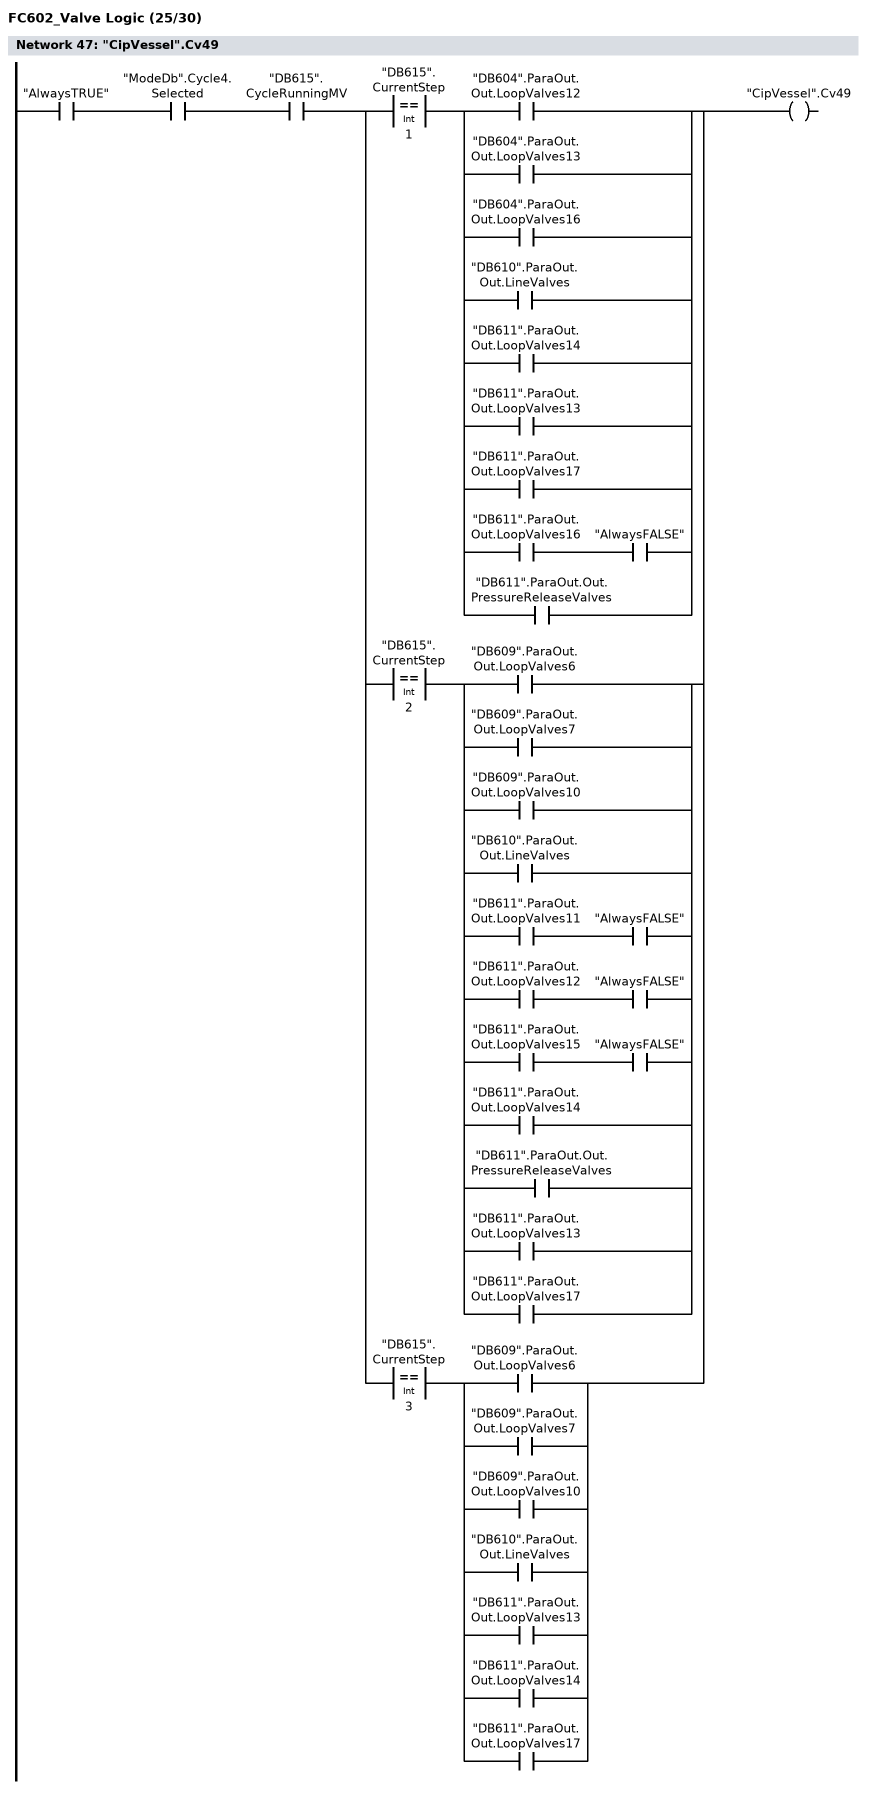
   RUNG wire#powerrail
      Contact( "AlwaysTRUE" )
      Contact( "ModeDb".Cycle4.Selected )
      Contact( "DB615".CycleRunningMV )
      wire#w1
      { S7_Templates := "SrcType := Int" } EQ_Contact(in1 := "DB615".CurrentStep, in2 := 1)
      wire#w2
      Contact( "DB604".ParaOut.Out.LoopValves12 )
      wire#w3
      Coil( "CipVessel".Cv49 )
   END_RUNG
   RUNG wire#w2
      Contact( "DB604".ParaOut.Out.LoopValves13 )
   END_RUNG wire#w3
   RUNG wire#w2
      Contact( "DB604".ParaOut.Out.LoopValves16 )
   END_RUNG wire#w3
   RUNG wire#w2
      Contact( "DB610".ParaOut.Out.LineValves )
   END_RUNG wire#w3
   RUNG wire#w2
      Contact( "DB611".ParaOut.Out.LoopValves14 )
   END_RUNG wire#w3
   RUNG wire#w2
      Contact( "DB611".ParaOut.Out.LoopValves13 )
   END_RUNG wire#w3
   RUNG wire#w2
      Contact( "DB611".ParaOut.Out.LoopValves17 )
   END_RUNG wire#w3
   RUNG wire#w2
      Contact( "DB611".ParaOut.Out.LoopValves16 )
      Contact( "AlwaysFALSE" )
   END_RUNG wire#w3
   RUNG wire#w2
      Contact( "DB611".ParaOut.Out.PressureReleaseValves )
   END_RUNG wire#w3
   RUNG wire#w1
      { S7_Templates := "SrcType := Int" } EQ_Contact(in1 := "DB615".CurrentStep, in2 := 2)
      wire#w4
      Contact( "DB609".ParaOut.Out.LoopValves6 )
   END_RUNG wire#w3
   RUNG wire#w4
      Contact( "DB609".ParaOut.Out.LoopValves7 )
   END_RUNG wire#w3
   RUNG wire#w4
      Contact( "DB609".ParaOut.Out.LoopValves10 )
   END_RUNG wire#w3
   RUNG wire#w4
      Contact( "DB610".ParaOut.Out.LineValves )
   END_RUNG wire#w3
   RUNG wire#w4
      Contact( "DB611".ParaOut.Out.LoopValves11 )
      Contact( "AlwaysFALSE" )
   END_RUNG wire#w3
   RUNG wire#w4
      Contact( "DB611".ParaOut.Out.LoopValves12 )
      Contact( "AlwaysFALSE" )
   END_RUNG wire#w3
   RUNG wire#w4
      Contact( "DB611".ParaOut.Out.LoopValves15 )
      Contact( "AlwaysFALSE" )
   END_RUNG wire#w3
   RUNG wire#w4
      Contact( "DB611".ParaOut.Out.LoopValves14 )
   END_RUNG wire#w3
   RUNG wire#w4
      Contact( "DB611".ParaOut.Out.PressureReleaseValves )
   END_RUNG wire#w3
   RUNG wire#w4
      Contact( "DB611".ParaOut.Out.LoopValves13 )
   END_RUNG wire#w3
   RUNG wire#w4
      Contact( "DB611".ParaOut.Out.LoopValves17 )
   END_RUNG wire#w3
   RUNG wire#w1
      { S7_Templates := "SrcType := Int" } EQ_Contact(in1 := "DB615".CurrentStep, in2 := 3)
      wire#w5
      Contact( "DB609".ParaOut.Out.LoopValves6 )
   END_RUNG wire#w3
   RUNG wire#w5
      Contact( "DB609".ParaOut.Out.LoopValves7 )
   END_RUNG wire#w3
   RUNG wire#w5
      Contact( "DB609".ParaOut.Out.LoopValves10 )
   END_RUNG wire#w3
   RUNG wire#w5
      Contact( "DB610".ParaOut.Out.LineValves )
   END_RUNG wire#w3
   RUNG wire#w5
      Contact( "DB611".ParaOut.Out.LoopValves13 )
   END_RUNG wire#w3
   RUNG wire#w5
      Contact( "DB611".ParaOut.Out.LoopValves14 )
   END_RUNG wire#w3
   RUNG wire#w5
      Contact( "DB611".ParaOut.Out.LoopValves17 )
   END_RUNG wire#w3
   // the same network as SCL:
   "CipVessel".Cv49 := "AlwaysTRUE" AND "ModeDb".Cycle4.Selected AND "DB615".CycleRunningMV AND ((("DB615".CurrentStep = 1) AND ("DB604".ParaOut.Out.LoopValves12 OR "DB604".ParaOut.Out.LoopValves13 OR "DB604".ParaOut.Out.LoopValves16 OR "DB610".ParaOut.Out.LineValves OR "DB611".ParaOut.Out.LoopValves14 OR "DB611".ParaOut.Out.LoopValves13 OR "DB611".ParaOut.Out.LoopValves17 OR ("DB611".ParaOut.Out.LoopValves16 AND "AlwaysFALSE") OR "DB611".ParaOut.Out.PressureReleaseValves)) OR (("DB615".CurrentStep = 2) AND ("DB609".ParaOut.Out.LoopValves6 OR "DB609".ParaOut.Out.LoopValves7 OR "DB609".ParaOut.Out.LoopValves10 OR "DB610".ParaOut.Out.LineValves OR ("DB611".ParaOut.Out.LoopValves11 AND "AlwaysFALSE") OR ("DB611".ParaOut.Out.LoopValves12 AND "AlwaysFALSE") OR ("DB611".ParaOut.Out.LoopValves15 AND "AlwaysFALSE") OR "DB611".ParaOut.Out.LoopValves14 OR "DB611".ParaOut.Out.PressureReleaseValves OR "DB611".ParaOut.Out.LoopValves13 OR "DB611".ParaOut.Out.LoopValves17)) OR (("DB615".CurrentStep = 3) AND ("DB609".ParaOut.Out.LoopValves6 OR "DB609".ParaOut.Out.LoopValves7 OR "DB609".ParaOut.Out.LoopValves10 OR "DB610".ParaOut.Out.LineValves OR "DB611".ParaOut.Out.LoopValves13 OR "DB611".ParaOut.Out.LoopValves14 OR "DB611".ParaOut.Out.LoopValves17)));
END_REGION

REGION Network 48: "CipVessel".Cv53
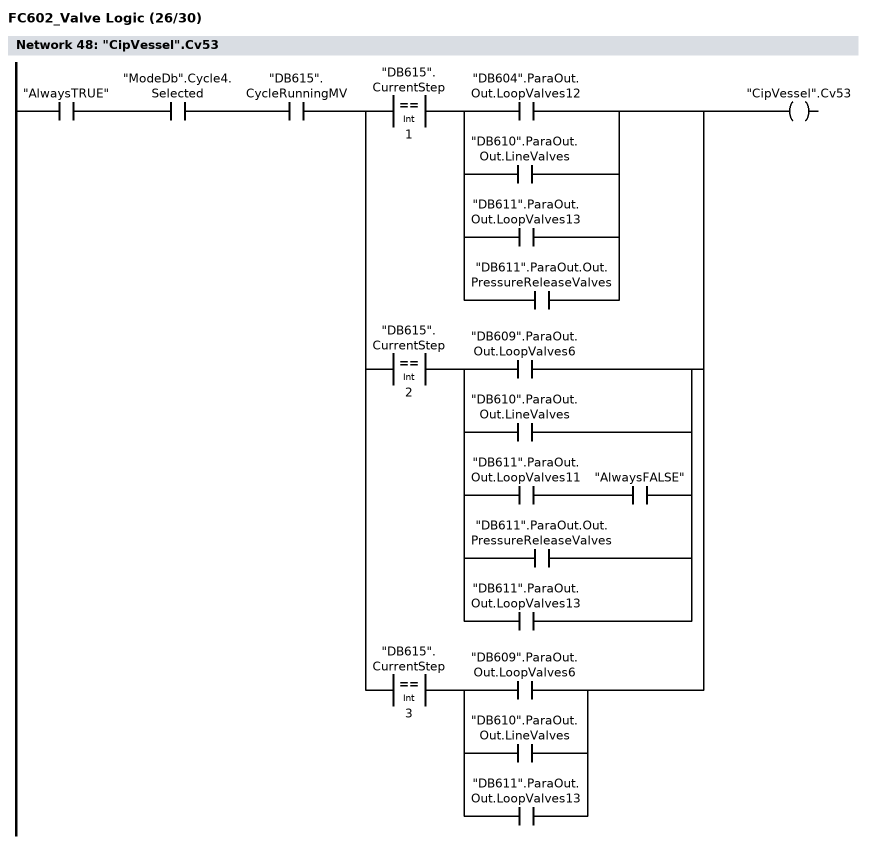
   RUNG wire#powerrail
      Contact( "AlwaysTRUE" )
      Contact( "ModeDb".Cycle4.Selected )
      Contact( "DB615".CycleRunningMV )
      wire#w1
      { S7_Templates := "SrcType := Int" } EQ_Contact(in1 := "DB615".CurrentStep, in2 := 1)
      wire#w2
      Contact( "DB604".ParaOut.Out.LoopValves12 )
      wire#w3
      Coil( "CipVessel".Cv53 )
   END_RUNG
   RUNG wire#w2
      Contact( "DB610".ParaOut.Out.LineValves )
   END_RUNG wire#w3
   RUNG wire#w2
      Contact( "DB611".ParaOut.Out.LoopValves13 )
   END_RUNG wire#w3
   RUNG wire#w2
      Contact( "DB611".ParaOut.Out.PressureReleaseValves )
   END_RUNG wire#w3
   RUNG wire#w1
      { S7_Templates := "SrcType := Int" } EQ_Contact(in1 := "DB615".CurrentStep, in2 := 2)
      wire#w4
      Contact( "DB609".ParaOut.Out.LoopValves6 )
   END_RUNG wire#w3
   RUNG wire#w4
      Contact( "DB610".ParaOut.Out.LineValves )
   END_RUNG wire#w3
   RUNG wire#w4
      Contact( "DB611".ParaOut.Out.LoopValves11 )
      Contact( "AlwaysFALSE" )
   END_RUNG wire#w3
   RUNG wire#w4
      Contact( "DB611".ParaOut.Out.PressureReleaseValves )
   END_RUNG wire#w3
   RUNG wire#w4
      Contact( "DB611".ParaOut.Out.LoopValves13 )
   END_RUNG wire#w3
   RUNG wire#w1
      { S7_Templates := "SrcType := Int" } EQ_Contact(in1 := "DB615".CurrentStep, in2 := 3)
      wire#w5
      Contact( "DB609".ParaOut.Out.LoopValves6 )
   END_RUNG wire#w3
   RUNG wire#w5
      Contact( "DB610".ParaOut.Out.LineValves )
   END_RUNG wire#w3
   RUNG wire#w5
      Contact( "DB611".ParaOut.Out.LoopValves13 )
   END_RUNG wire#w3
   // the same network as SCL:
   "CipVessel".Cv53 := "AlwaysTRUE" AND "ModeDb".Cycle4.Selected AND "DB615".CycleRunningMV AND ((("DB615".CurrentStep = 1) AND ("DB604".ParaOut.Out.LoopValves12 OR "DB610".ParaOut.Out.LineValves OR "DB611".ParaOut.Out.LoopValves13 OR "DB611".ParaOut.Out.PressureReleaseValves)) OR (("DB615".CurrentStep = 2) AND ("DB609".ParaOut.Out.LoopValves6 OR "DB610".ParaOut.Out.LineValves OR ("DB611".ParaOut.Out.LoopValves11 AND "AlwaysFALSE") OR "DB611".ParaOut.Out.PressureReleaseValves OR "DB611".ParaOut.Out.LoopValves13)) OR (("DB615".CurrentStep = 3) AND ("DB609".ParaOut.Out.LoopValves6 OR "DB610".ParaOut.Out.LineValves OR "DB611".ParaOut.Out.LoopValves13)));
END_REGION

REGION Network 49: ----------- PF02 OUT -------------
END_REGION

REGION Network 50: "CipVessel".Cv56
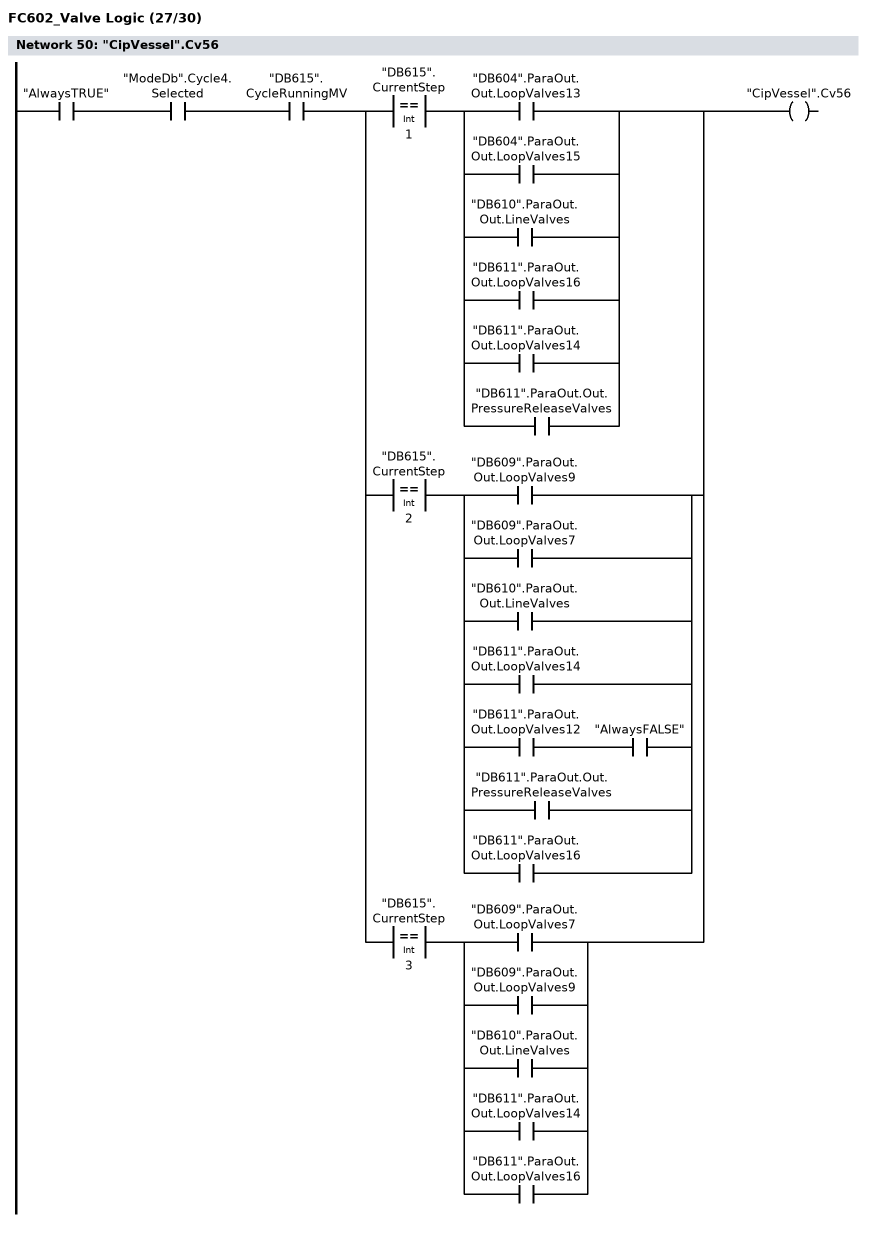
   RUNG wire#powerrail
      Contact( "AlwaysTRUE" )
      Contact( "ModeDb".Cycle4.Selected )
      Contact( "DB615".CycleRunningMV )
      wire#w1
      { S7_Templates := "SrcType := Int" } EQ_Contact(in1 := "DB615".CurrentStep, in2 := 1)
      wire#w2
      Contact( "DB604".ParaOut.Out.LoopValves13 )
      wire#w3
      Coil( "CipVessel".Cv56 )
   END_RUNG
   RUNG wire#w2
      Contact( "DB604".ParaOut.Out.LoopValves15 )
   END_RUNG wire#w3
   RUNG wire#w2
      Contact( "DB610".ParaOut.Out.LineValves )
   END_RUNG wire#w3
   RUNG wire#w2
      Contact( "DB611".ParaOut.Out.LoopValves16 )
   END_RUNG wire#w3
   RUNG wire#w2
      Contact( "DB611".ParaOut.Out.LoopValves14 )
   END_RUNG wire#w3
   RUNG wire#w2
      Contact( "DB611".ParaOut.Out.PressureReleaseValves )
   END_RUNG wire#w3
   RUNG wire#w1
      { S7_Templates := "SrcType := Int" } EQ_Contact(in1 := "DB615".CurrentStep, in2 := 2)
      wire#w4
      Contact( "DB609".ParaOut.Out.LoopValves9 )
   END_RUNG wire#w3
   RUNG wire#w4
      Contact( "DB609".ParaOut.Out.LoopValves7 )
   END_RUNG wire#w3
   RUNG wire#w4
      Contact( "DB610".ParaOut.Out.LineValves )
   END_RUNG wire#w3
   RUNG wire#w4
      Contact( "DB611".ParaOut.Out.LoopValves14 )
   END_RUNG wire#w3
   RUNG wire#w4
      Contact( "DB611".ParaOut.Out.LoopValves12 )
      Contact( "AlwaysFALSE" )
   END_RUNG wire#w3
   RUNG wire#w4
      Contact( "DB611".ParaOut.Out.PressureReleaseValves )
   END_RUNG wire#w3
   RUNG wire#w4
      Contact( "DB611".ParaOut.Out.LoopValves16 )
   END_RUNG wire#w3
   RUNG wire#w1
      { S7_Templates := "SrcType := Int" } EQ_Contact(in1 := "DB615".CurrentStep, in2 := 3)
      wire#w5
      Contact( "DB609".ParaOut.Out.LoopValves7 )
   END_RUNG wire#w3
   RUNG wire#w5
      Contact( "DB609".ParaOut.Out.LoopValves9 )
   END_RUNG wire#w3
   RUNG wire#w5
      Contact( "DB610".ParaOut.Out.LineValves )
   END_RUNG wire#w3
   RUNG wire#w5
      Contact( "DB611".ParaOut.Out.LoopValves14 )
   END_RUNG wire#w3
   RUNG wire#w5
      Contact( "DB611".ParaOut.Out.LoopValves16 )
   END_RUNG wire#w3
   // the same network as SCL:
   "CipVessel".Cv56 := "AlwaysTRUE" AND "ModeDb".Cycle4.Selected AND "DB615".CycleRunningMV AND ((("DB615".CurrentStep = 1) AND ("DB604".ParaOut.Out.LoopValves13 OR "DB604".ParaOut.Out.LoopValves15 OR "DB610".ParaOut.Out.LineValves OR "DB611".ParaOut.Out.LoopValves16 OR "DB611".ParaOut.Out.LoopValves14 OR "DB611".ParaOut.Out.PressureReleaseValves)) OR (("DB615".CurrentStep = 2) AND ("DB609".ParaOut.Out.LoopValves9 OR "DB609".ParaOut.Out.LoopValves7 OR "DB610".ParaOut.Out.LineValves OR "DB611".ParaOut.Out.LoopValves14 OR ("DB611".ParaOut.Out.LoopValves12 AND "AlwaysFALSE") OR "DB611".ParaOut.Out.PressureReleaseValves OR "DB611".ParaOut.Out.LoopValves16)) OR (("DB615".CurrentStep = 3) AND ("DB609".ParaOut.Out.LoopValves7 OR "DB609".ParaOut.Out.LoopValves9 OR "DB610".ParaOut.Out.LineValves OR "DB611".ParaOut.Out.LoopValves14 OR "DB611".ParaOut.Out.LoopValves16)));
END_REGION

REGION Network 51: "CipVessel".Cv57
